LIN {X 0,Y 496.772,Z 250.855,A -85,B 0,C 180,E1 18209.944,E2 18209.944} C_VEL
LIN {X 0,Y 496.758,Z 250.853,A -85,B 0,C 180,E1 18206.403,E2 18206.403} C_VEL
LIN {X 0,Y 496.769,Z 250.851,A -85,B 0,C 180,E1 18202.804,E2 18202.804} C_VEL
LIN {X 0,Y 496.753,Z 250.856,A -85,B 0,C 180,E1 18199.264,E2 18199.264} C_VEL
LIN {X 0,Y 496.754,Z 250.857,A -85,B 0,C 180,E1 18195.648,E2 18195.648} C_VEL
LIN {X 0,Y 496.767,Z 250.857,A -85,B 0,C 180,E1 18192.084,E2 18192.084} C_VEL
LIN {X 0,Y 496.769,Z 250.855,A -85,B 0,C 180,E1 18188.45,E2 18188.45} C_VEL
LIN {X 0,Y 496.745,Z 250.851,A -85,B 0,C 180,E1 18184.966,E2 18184.966} C_VEL
LIN {X 0,Y 496.736,Z 250.854,A -85,B 0,C 180,E1 18181.385,E2 18181.385} C_VEL
LIN {X 0,Y 496.764,Z 250.853,A -85,B 0,C 180,E1 18177.925,E2 18177.925} C_VEL
LIN {X 0,Y 496.768,Z 250.855,A -85,B 0,C 180,E1 18174.341,E2 18174.341} C_VEL
LIN {X 0,Y 496.725,Z 250.858,A -85,B 0,C 180,E1 18170.968,E2 18170.968} C_VEL
LIN {X 0,Y 496.723,Z 250.861,A -85,B 0,C 180,E1 18167.327,E2 18167.327} C_VEL
LIN {X 0,Y 496.769,Z 250.856,A -85,B 0,C 180,E1 18163.995,E2 18163.995} C_VEL
LIN {X 0,Y 496.736,Z 250.862,A -85,B 0,C 180,E1 18160.481,E2 18160.481} C_VEL
LIN {X 0,Y 496.706,Z 250.846,A -85,B 0,C 180,E1 18157.015,E2 18157.015} C_VEL
LIN {X 0,Y 496.788,Z 251.097,A -85,B 0,C 180,E1 18155.823,E2 18155.823} C_VEL
LIN {X 0,Y 498.222,Z 254.643,A -85,B 0,C 180,E1 18155.266,E2 18155.266} C_VEL
LIN {X 0,Y 505.949,Z 273.047,A -85,B 0,C 180,E1 18152.712,E2 18152.712} C_VEL
LIN {X 0,Y 509.561,Z 282.883,A -85,B 0,C 180,E1 18151.46,E2 18151.46} C_VEL
LIN {X 0,Y 508.599,Z 300.101,A -85,B 0,C 180,E1 18150.013,E2 18150.013} C_VEL
LIN {X 0,Y 512.119,Z 319.644,A -85,B 0,C 180,E1 18149.37,E2 18149.37} C_VEL
LIN {X 0,Y 509.717,Z 467.45,A -85,B 0,C 180,E1 18147.041,E2 18147.041} C_VEL
LIN {X 0,Y 508.732,Z 475.141,A -85,B 0,C 180,E1 18146.984,E2 18146.984} C_VEL
LIN {X 0,Y 503.194,Z 495.645,A -85,B 0,C 180,E1 18147.05,E2 18147.05} C_VEL
LIN {X 0,Y 502.468,Z 502.242,A -85,B 0,C 180,E1 18146.991,E2 18146.991} C_VEL
LIN {X 0,Y 501.359,Z 564.042,A -85,B 0,C 180,E1 18145.978,E2 18145.978} C_VEL
LIN {X 0,Y 500.552,Z 584.976,A -85,B 0,C 180,E1 18145.421,E2 18145.421} C_VEL
LIN {X 0,Y 499.562,Z 604.152,A -85,B 0,C 180,E1 18144.698,E2 18144.698} C_VEL
LIN {X 0,Y 498.327,Z 623.36,A -85,B 0,C 180,E1 18143.765,E2 18143.765} C_VEL
LIN {X 0,Y 496.896,Z 642.75,A -85,B 0,C 180,E1 18142.579,E2 18142.579} C_VEL
LIN {X 0,Y 495.485,Z 660.162,A -85,B 0,C 180,E1 18141.279,E2 18141.279} C_VEL
LIN {X 0,Y 494.046,Z 676.802,A -85,B 0,C 180,E1 18139.792,E2 18139.792} C_VEL
LIN {X 0,Y 492.609,Z 692.858,A -85,B 0,C 180,E1 18138.074,E2 18138.074} C_VEL
LIN {X 0,Y 491.318,Z 707.439,A -85,B 0,C 180,E1 18136.22,E2 18136.22} C_VEL
LIN {X 0,Y 490.214,Z 720.639,A -85,B 0,C 180,E1 18134.232,E2 18134.232} C_VEL
LIN {X 0,Y 489.314,Z 733.716,A -85,B 0,C 180,E1 18131.928,E2 18131.928} C_VEL
LIN {X 0,Y 488.706,Z 744.41,A -85,B 0,C 180,E1 18129.668,E2 18129.668} C_VEL
LIN {X 0,Y 488.303,Z 753.506,A -85,B 0,C 180,E1 18127.309,E2 18127.309} C_VEL
LIN {X 0,Y 488.069,Z 760.637,A -85,B 0,C 180,E1 18124.974,E2 18124.974} C_VEL
LIN {X 0,Y 487.961,Z 766.109,A -85,B 0,C 180,E1 18122.61,E2 18122.61} C_VEL
LIN {X 0,Y 487.919,Z 769.788,A -85,B 0,C 180,E1 18120.273,E2 18120.273} C_VEL
LIN {X 0,Y 487.914,Z 771.861,A -85,B 0,C 180,E1 18117.97,E2 18117.97} C_VEL
LIN {X 0,Y 487.908,Z 772.443,A -85,B 0,C 180,E1 18115.621,E2 18115.621} C_VEL
LIN {X 0,Y 487.916,Z 771.488,A -85,B 0,C 180,E1 18113.298,E2 18113.298} C_VEL
LIN {X 0,Y 487.926,Z 768.745,A -85,B 0,C 180,E1 18110.868,E2 18110.868} C_VEL
LIN {X 0,Y 487.978,Z 764.447,A -85,B 0,C 180,E1 18108.518,E2 18108.518} C_VEL
LIN {X 0,Y 488.144,Z 758.138,A -85,B 0,C 180,E1 18106.054,E2 18106.054} C_VEL
LIN {X 0,Y 488.428,Z 750.424,A -85,B 0,C 180,E1 18103.738,E2 18103.738} C_VEL
LIN {X 0,Y 488.861,Z 741.482,A -85,B 0,C 180,E1 18101.564,E2 18101.564} C_VEL
LIN {X 0,Y 489.546,Z 730.05,A -85,B 0,C 180,E1 18099.286,E2 18099.286} C_VEL
LIN {X 0,Y 490.601,Z 715.79,A -85,B 0,C 180,E1 18096.907,E2 18096.907} C_VEL
LIN {X 0,Y 491.817,Z 701.453,A -85,B 0,C 180,E1 18094.899,E2 18094.899} C_VEL
LIN {X 0,Y 493.162,Z 685.95,A -85,B 0,C 180,E1 18093.081,E2 18093.081} C_VEL
LIN {X 0,Y 494.552,Z 669.994,A -85,B 0,C 180,E1 18091.507,E2 18091.507} C_VEL
LIN {X 0,Y 495.957,Z 653.26,A -85,B 0,C 180,E1 18090.117,E2 18090.117} C_VEL
LIN {X 0,Y 497.377,Z 634.922,A -85,B 0,C 180,E1 18088.849,E2 18088.849} C_VEL
LIN {X 0,Y 498.675,Z 616.606,A -85,B 0,C 180,E1 18087.818,E2 18087.818} C_VEL
LIN {X 0,Y 499.814,Z 596.729,A -85,B 0,C 180,E1 18086.934,E2 18086.934} C_VEL
LIN {X 0,Y 500.752,Z 576.616,A -85,B 0,C 180,E1 18086.273,E2 18086.273} C_VEL
LIN {X 0,Y 501.378,Z 555.957,A -85,B 0,C 180,E1 18085.807,E2 18085.807} C_VEL
LIN {X 0,Y 505.231,Z 320.117,A -85,B 0,C 180,E1 18082.071,E2 18082.071} C_VEL
LIN {X 0,Y 501.409,Z 299.001,A -85,B 0,C 180,E1 18081.342,E2 18081.342} C_VEL
LIN {X 0,Y 502.22,Z 285.202,A -85,B 0,C 180,E1 18080.143,E2 18080.143} C_VEL
LIN {X 0,Y 494.741,Z 266.119,A -85,B 0,C 180,E1 18077.631,E2 18077.631} C_VEL
LIN {X 0,Y 488.853,Z 252.1,A -85,B 0,C 180,E1 18075.612,E2 18075.612} C_VEL
LIN {X 0,Y 488.818,Z 251.843,A -85,B 0,C 180,E1 18073.595,E2 18073.595} C_VEL
LIN {X 0,Y 488.826,Z 251.834,A -85,B 0,C 180,E1 18070.028,E2 18070.028} C_VEL
LIN {X 0,Y 488.824,Z 251.807,A -85,B 0,C 180,E1 18066.367,E2 18066.367} C_VEL
LIN {X 0,Y 488.822,Z 251.844,A -85,B 0,C 180,E1 18062.732,E2 18062.732} C_VEL
LIN {X 0,Y 488.81,Z 251.842,A -85,B 0,C 180,E1 18059.11,E2 18059.11} C_VEL
LIN {X 0,Y 488.822,Z 251.842,A -85,B 0,C 180,E1 18055.489,E2 18055.489} C_VEL
LIN {X 0,Y 488.827,Z 251.847,A -85,B 0,C 180,E1 18051.852,E2 18051.852} C_VEL
LIN {X 0,Y 488.831,Z 251.841,A -85,B 0,C 180,E1 18048.292,E2 18048.292} C_VEL
LIN {X 0,Y 488.81,Z 251.841,A -85,B 0,C 180,E1 18044.718,E2 18044.718} C_VEL
LIN {X 0,Y 488.819,Z 251.833,A -85,B 0,C 180,E1 18041.175,E2 18041.175} C_VEL
LIN {X 0,Y 488.828,Z 251.845,A -85,B 0,C 180,E1 18037.67,E2 18037.67} C_VEL
LIN {X 0,Y 488.825,Z 251.839,A -85,B 0,C 180,E1 18034.069,E2 18034.069} C_VEL
LIN {X 0,Y 488.808,Z 251.833,A -85,B 0,C 180,E1 18030.481,E2 18030.481} C_VEL
LIN {X 0,Y 488.813,Z 251.841,A -85,B 0,C 180,E1 18026.874,E2 18026.874} C_VEL
LIN {X 0,Y 488.832,Z 251.841,A -85,B 0,C 180,E1 18023.25,E2 18023.25} C_VEL
LIN {X 0,Y 488.828,Z 251.829,A -85,B 0,C 180,E1 18019.598,E2 18019.598} C_VEL
LIN {X 0,Y 488.812,Z 251.841,A -85,B 0,C 180,E1 18016.029,E2 18016.029} C_VEL
LIN {X 0,Y 488.804,Z 251.844,A -85,B 0,C 180,E1 18012.401,E2 18012.401} C_VEL
LIN {X 0,Y 488.821,Z 251.832,A -85,B 0,C 180,E1 18008.823,E2 18008.823} C_VEL
LIN {X 0,Y 488.829,Z 251.844,A -85,B 0,C 180,E1 18005.28,E2 18005.28} C_VEL
LIN {X 0,Y 488.822,Z 251.835,A -85,B 0,C 180,E1 18001.64,E2 18001.64} C_VEL
LIN {X 0,Y 488.802,Z 251.832,A -85,B 0,C 180,E1 17998.124,E2 17998.124} C_VEL
LIN {X 0,Y 488.82,Z 251.845,A -85,B 0,C 180,E1 17994.6,E2 17994.6} C_VEL
LIN {X 0,Y 488.83,Z 251.837,A -85,B 0,C 180,E1 17991.056,E2 17991.056} C_VEL
LIN {X 0,Y 488.814,Z 251.829,A -85,B 0,C 180,E1 17987.477,E2 17987.477} C_VEL
LIN {X 0,Y 488.8,Z 251.839,A -85,B 0,C 180,E1 17983.969,E2 17983.969} C_VEL
LIN {X 0,Y 488.82,Z 251.845,A -85,B 0,C 180,E1 17980.399,E2 17980.399} C_VEL
LIN {X 0,Y 488.832,Z 251.844,A -85,B 0,C 180,E1 17976.876,E2 17976.876} C_VEL
LIN {X 0,Y 488.815,Z 251.844,A -85,B 0,C 180,E1 17973.255,E2 17973.255} C_VEL
LIN {X 0,Y 488.799,Z 251.848,A -85,B 0,C 180,E1 17969.676,E2 17969.676} C_VEL
LIN {X 0,Y 488.817,Z 251.847,A -85,B 0,C 180,E1 17966.143,E2 17966.143} C_VEL
LIN {X 0,Y 488.833,Z 251.84,A -85,B 0,C 180,E1 17962.522,E2 17962.522} C_VEL
LIN {X 0,Y 488.819,Z 251.84,A -85,B 0,C 180,E1 17958.959,E2 17958.959} C_VEL
LIN {X 0,Y 488.808,Z 251.913,A -85,B 0,C 180,E1 17955.549,E2 17955.549} C_VEL
LIN {X 0,Y 489.229,Z 253.594,A -85,B 0,C 180,E1 17955.245,E2 17955.245} C_VEL
LIN {X 0,Y 492.865,Z 260.965,A -85,B 0,C 180,E1 17954.253,E2 17954.253} C_VEL
LIN {X 0,Y 501.354,Z 279.391,A -85,B 0,C 180,E1 17951.937,E2 17951.937} C_VEL
LIN {X 0,Y 506.352,Z 291.141,A -85,B 0,C 180,E1 17950.588,E2 17950.588} C_VEL
LIN {X 0,Y 505.835,Z 302.61,A -85,B 0,C 180,E1 17949.815,E2 17949.815} C_VEL
LIN {X 0,Y 509.159,Z 324.69,A -85,B 0,C 180,E1 17949.147,E2 17949.147} C_VEL
LIN {X 0,Y 505.913,Z 541.603,A -85,B 0,C 180,E1 17945.733,E2 17945.733} C_VEL
LIN {X 0,Y 504.85,Z 609.184,A -85,B 0,C 180,E1 17944.654,E2 17944.654} C_VEL
LIN {X 0,Y 503.96,Z 630.518,A -85,B 0,C 180,E1 17944.117,E2 17944.117} C_VEL
LIN {X 0,Y 502.77,Z 653.144,A -85,B 0,C 180,E1 17943.329,E2 17943.329} C_VEL
LIN {X 0,Y 501.528,Z 673.269,A -85,B 0,C 180,E1 17942.429,E2 17942.429} C_VEL
LIN {X 0,Y 500.051,Z 692.001,A -85,B 0,C 180,E1 17941.373,E2 17941.373} C_VEL
LIN {X 0,Y 498.309,Z 712.512,A -85,B 0,C 180,E1 17939.973,E2 17939.973} C_VEL
LIN {X 0,Y 496.643,Z 730.768,A -85,B 0,C 180,E1 17938.497,E2 17938.497} C_VEL
LIN {X 0,Y 494.933,Z 748.878,A -85,B 0,C 180,E1 17936.757,E2 17936.757} C_VEL
LIN {X 0,Y 493.327,Z 765.681,A -85,B 0,C 180,E1 17934.868,E2 17934.868} C_VEL
LIN {X 0,Y 491.919,Z 781.186,A -85,B 0,C 180,E1 17932.842,E2 17932.842} C_VEL
LIN {X 0,Y 490.705,Z 795.639,A -85,B 0,C 180,E1 17930.639,E2 17930.639} C_VEL
LIN {X 0,Y 489.724,Z 808.46,A -85,B 0,C 180,E1 17928.324,E2 17928.324} C_VEL
LIN {X 0,Y 488.981,Z 819.817,A -85,B 0,C 180,E1 17925.901,E2 17925.901} C_VEL
LIN {X 0,Y 488.485,Z 829.264,A -85,B 0,C 180,E1 17923.492,E2 17923.492} C_VEL
LIN {X 0,Y 488.176,Z 836.886,A -85,B 0,C 180,E1 17921.099,E2 17921.099} C_VEL
LIN {X 0,Y 488.003,Z 843.148,A -85,B 0,C 180,E1 17918.601,E2 17918.601} C_VEL
LIN {X 0,Y 487.936,Z 847.824,A -85,B 0,C 180,E1 17916.116,E2 17916.116} C_VEL
LIN {X 0,Y 487.907,Z 850.804,A -85,B 0,C 180,E1 17913.625,E2 17913.625} C_VEL
LIN {X 0,Y 487.911,Z 852.305,A -85,B 0,C 180,E1 17911.056,E2 17911.056} C_VEL
LIN {X 0,Y 487.906,Z 852.258,A -85,B 0,C 180,E1 17908.707,E2 17908.707} C_VEL
LIN {X 0,Y 487.908,Z 850.67,A -85,B 0,C 180,E1 17906.239,E2 17906.239} C_VEL
LIN {X 0,Y 487.938,Z 847.63,A -85,B 0,C 180,E1 17903.764,E2 17903.764} C_VEL
LIN {X 0,Y 488.004,Z 843.142,A -85,B 0,C 180,E1 17901.397,E2 17901.397} C_VEL
LIN {X 0,Y 488.184,Z 836.668,A -85,B 0,C 180,E1 17898.828,E2 17898.828} C_VEL
LIN {X 0,Y 488.509,Z 828.845,A -85,B 0,C 180,E1 17896.385,E2 17896.385} C_VEL
LIN {X 0,Y 489.028,Z 819.123,A -85,B 0,C 180,E1 17893.936,E2 17893.936} C_VEL
LIN {X 0,Y 489.771,Z 807.812,A -85,B 0,C 180,E1 17891.552,E2 17891.552} C_VEL
LIN {X 0,Y 490.706,Z 795.623,A -85,B 0,C 180,E1 17889.358,E2 17889.358} C_VEL
LIN {X 0,Y 491.921,Z 781.168,A -85,B 0,C 180,E1 17887.155,E2 17887.155} C_VEL
LIN {X 0,Y 493.328,Z 765.66,A -85,B 0,C 180,E1 17885.129,E2 17885.129} C_VEL
LIN {X 0,Y 494.949,Z 748.687,A -85,B 0,C 180,E1 17883.224,E2 17883.224} C_VEL
LIN {X 0,Y 496.646,Z 730.741,A -85,B 0,C 180,E1 17881.501,E2 17881.501} C_VEL
LIN {X 0,Y 498.312,Z 712.484,A -85,B 0,C 180,E1 17880.024,E2 17880.024} C_VEL
LIN {X 0,Y 500.053,Z 691.996,A -85,B 0,C 180,E1 17878.626,E2 17878.626} C_VEL
LIN {X 0,Y 501.531,Z 673.215,A -85,B 0,C 180,E1 17877.568,E2 17877.568} C_VEL
LIN {X 0,Y 502.804,Z 652.224,A -85,B 0,C 180,E1 17876.637,E2 17876.637} C_VEL
LIN {X 0,Y 503.967,Z 629.777,A -85,B 0,C 180,E1 17875.868,E2 17875.868} C_VEL
LIN {X 0,Y 504.829,Z 608.318,A -85,B 0,C 180,E1 17875.337,E2 17875.337} C_VEL
LIN {X 0,Y 506.756,Z 476.023,A -85,B 0,C 180,E1 17873.262,E2 17873.262} C_VEL
LIN {X 0,Y 508.836,Z 322.634,A -85,B 0,C 180,E1 17870.839,E2 17870.839} C_VEL
LIN {X 0,Y 505.54,Z 301.596,A -85,B 0,C 180,E1 17870.184,E2 17870.184} C_VEL
LIN {X 0,Y 505.959,Z 290.005,A -85,B 0,C 180,E1 17869.363,E2 17869.363} C_VEL
LIN {X 0,Y 495.083,Z 265.808,A -85,B 0,C 180,E1 17866.472,E2 17866.472} C_VEL
LIN {X 0,Y 490.052,Z 255.211,A -85,B 0,C 180,E1 17865.072,E2 17865.072} C_VEL
LIN {X 0,Y 488.846,Z 252.112,A -85,B 0,C 180,E1 17864.619,E2 17864.619} C_VEL
LIN {X 0,Y 488.829,Z 251.842,A -85,B 0,C 180,E1 17861.508,E2 17861.508} C_VEL
LIN {X 0,Y 488.83,Z 251.844,A -85,B 0,C 180,E1 17857.852,E2 17857.852} C_VEL
LIN {X 0,Y 488.82,Z 251.844,A -85,B 0,C 180,E1 17854.229,E2 17854.229} C_VEL
LIN {X 0,Y 488.818,Z 251.844,A -85,B 0,C 180,E1 17850.619,E2 17850.619} C_VEL
LIN {X 0,Y 488.829,Z 251.841,A -85,B 0,C 180,E1 17847.007,E2 17847.007} C_VEL
LIN {X 0,Y 488.816,Z 251.841,A -85,B 0,C 180,E1 17843.38,E2 17843.38} C_VEL
LIN {X 0,Y 488.823,Z 251.844,A -85,B 0,C 180,E1 17839.795,E2 17839.795} C_VEL
LIN {X 0,Y 488.828,Z 251.844,A -85,B 0,C 180,E1 17836.152,E2 17836.152} C_VEL
LIN {X 0,Y 488.83,Z 251.844,A -85,B 0,C 180,E1 17832.523,E2 17832.523} C_VEL
LIN {X 0,Y 488.815,Z 251.843,A -85,B 0,C 180,E1 17828.895,E2 17828.895} C_VEL
LIN {X 0,Y 488.801,Z 251.843,A -85,B 0,C 180,E1 17825.4,E2 17825.4} C_VEL
LIN {X 0,Y 488.823,Z 251.841,A -85,B 0,C 180,E1 17821.876,E2 17821.876} C_VEL
LIN {X 0,Y 488.831,Z 251.839,A -85,B 0,C 180,E1 17818.36,E2 17818.36} C_VEL
LIN {X 0,Y 488.797,Z 251.845,A -85,B 0,C 180,E1 17814.837,E2 17814.837} C_VEL
LIN {X 0,Y 488.787,Z 251.849,A -85,B 0,C 180,E1 17811.295,E2 17811.295} C_VEL
LIN {X 0,Y 488.818,Z 251.843,A -85,B 0,C 180,E1 17807.839,E2 17807.839} C_VEL
LIN {X 0,Y 488.818,Z 251.848,A -85,B 0,C 180,E1 17804.337,E2 17804.337} C_VEL
LIN {X 0,Y 488.776,Z 251.852,A -85,B 0,C 180,E1 17800.896,E2 17800.896} C_VEL
LIN {X 0,Y 488.771,Z 251.834,A -85,B 0,C 180,E1 17797.256,E2 17797.256} C_VEL
LIN {X 0,Y 488.823,Z 252.135,A -85,B 0,C 180,E1 17796.59,E2 17796.59} C_VEL
LIN {X 0,Y 495.725,Z 268.342,A -85,B 0,C 180,E1 17794.174,E2 17794.174} C_VEL
LIN {X 0,Y 502.718,Z 285.823,A -85,B 0,C 180,E1 17791.814,E2 17791.814} C_VEL
LIN {X 0,Y 501.902,Z 300.091,A -85,B 0,C 180,E1 17790.599,E2 17790.599} C_VEL
LIN {X 0,Y 505.67,Z 321.039,A -85,B 0,C 180,E1 17789.889,E2 17789.889} C_VEL
LIN {X 0,Y 502.468,Z 502.242,A -85,B 0,C 180,E1 17786.991,E2 17786.991} C_VEL
LIN {X 0,Y 501.504,Z 509.932,A -85,B 0,C 180,E1 17786.932,E2 17786.932} C_VEL
LIN {X 0,Y 495.893,Z 530.424,A -85,B 0,C 180,E1 17787.002,E2 17787.002} C_VEL
LIN {X 0,Y 495.165,Z 537.023,A -85,B 0,C 180,E1 17786.942,E2 17786.942} C_VEL
LIN {X 0,Y 494.491,Z 566.986,A -85,B 0,C 180,E1 17786.409,E2 17786.409} C_VEL
LIN {X 0,Y 493.652,Z 587.312,A -85,B 0,C 180,E1 17785.84,E2 17785.84} C_VEL
LIN {X 0,Y 492.563,Z 606.745,A -85,B 0,C 180,E1 17785.082,E2 17785.082} C_VEL
LIN {X 0,Y 491.214,Z 625.979,A -85,B 0,C 180,E1 17784.109,E2 17784.109} C_VEL
LIN {X 0,Y 489.754,Z 644.17,A -85,B 0,C 180,E1 17782.964,E2 17782.964} C_VEL
LIN {X 0,Y 488.174,Z 662.153,A -85,B 0,C 180,E1 17781.585,E2 17781.585} C_VEL
LIN {X 0,Y 486.698,Z 677.989,A -85,B 0,C 180,E1 17780.138,E2 17780.138} C_VEL
LIN {X 0,Y 485.179,Z 693.746,A -85,B 0,C 180,E1 17778.425,E2 17778.425} C_VEL
LIN {X 0,Y 483.783,Z 708.188,A -85,B 0,C 180,E1 17776.559,E2 17776.559} C_VEL
LIN {X 0,Y 482.576,Z 721.36,A -85,B 0,C 180,E1 17774.544,E2 17774.544} C_VEL
LIN {X 0,Y 481.576,Z 733.418,A -85,B 0,C 180,E1 17772.345,E2 17772.345} C_VEL
LIN {X 0,Y 480.795,Z 744.555,A -85,B 0,C 180,E1 17769.884,E2 17769.884} C_VEL
LIN {X 0,Y 480.337,Z 753.727,A -85,B 0,C 180,E1 17767.433,E2 17767.433} C_VEL
LIN {X 0,Y 480.083,Z 760.779,A -85,B 0,C 180,E1 17765.069,E2 17765.069} C_VEL
LIN {X 0,Y 479.968,Z 766.157,A -85,B 0,C 180,E1 17762.693,E2 17762.693} C_VEL
LIN {X 0,Y 479.921,Z 769.878,A -85,B 0,C 180,E1 17760.278,E2 17760.278} C_VEL
LIN {X 0,Y 479.914,Z 771.889,A -85,B 0,C 180,E1 17757.953,E2 17757.953} C_VEL
LIN {X 0,Y 479.908,Z 772.43,A -85,B 0,C 180,E1 17755.549,E2 17755.549} C_VEL
LIN {X 0,Y 479.918,Z 771.439,A -85,B 0,C 180,E1 17753.19,E2 17753.19} C_VEL
LIN {X 0,Y 479.927,Z 768.645,A -85,B 0,C 180,E1 17750.708,E2 17750.708} C_VEL
LIN {X 0,Y 479.992,Z 764.32,A -85,B 0,C 180,E1 17748.334,E2 17748.334} C_VEL
LIN {X 0,Y 480.173,Z 758.026,A -85,B 0,C 180,E1 17745.849,E2 17745.849} C_VEL
LIN {X 0,Y 480.497,Z 750.218,A -85,B 0,C 180,E1 17743.478,E2 17743.478} C_VEL
LIN {X 0,Y 481.102,Z 739.711,A -85,B 0,C 180,E1 17740.903,E2 17740.903} C_VEL
LIN {X 0,Y 481.916,Z 728.949,A -85,B 0,C 180,E1 17738.713,E2 17738.713} C_VEL
LIN {X 0,Y 482.944,Z 716.915,A -85,B 0,C 180,E1 17736.659,E2 17736.659} C_VEL
LIN {X 0,Y 484.254,Z 702.628,A -85,B 0,C 180,E1 17734.62,E2 17734.62} C_VEL
LIN {X 0,Y 485.647,Z 687.74,A -85,B 0,C 180,E1 17732.833,E2 17732.833} C_VEL
LIN {X 0,Y 487.138,Z 672.001,A -85,B 0,C 180,E1 17731.236,E2 17731.236} C_VEL
LIN {X 0,Y 488.768,Z 654.028,A -85,B 0,C 180,E1 17729.708,E2 17729.708} C_VEL
LIN {X 0,Y 490.291,Z 635.723,A -85,B 0,C 180,E1 17728.424,E2 17728.424} C_VEL
LIN {X 0,Y 491.68,Z 617.468,A -85,B 0,C 180,E1 17727.379,E2 17727.379} C_VEL
LIN {X 0,Y 492.891,Z 597.642,A -85,B 0,C 180,E1 17726.483,E2 17726.483} C_VEL
LIN {X 0,Y 493.89,Z 577.709,A -85,B 0,C 180,E1 17725.815,E2 17725.815} C_VEL
LIN {X 0,Y 494.571,Z 556.973,A -85,B 0,C 180,E1 17725.334,E2 17725.334} C_VEL
LIN {X 0,Y 498.755,Z 321.538,A -85,B 0,C 180,E1 17721.55,E2 17721.55} C_VEL
LIN {X 0,Y 494.681,Z 298.995,A -85,B 0,C 180,E1 17720.755,E2 17720.755} C_VEL
LIN {X 0,Y 495.303,Z 288.494,A -85,B 0,C 180,E1 17719.828,E2 17719.828} C_VEL
LIN {X 0,Y 488.224,Z 270.414,A -85,B 0,C 180,E1 17717.404,E2 17717.404} C_VEL
LIN {X 0,Y 482.117,Z 256.202,A -85,B 0,C 180,E1 17715.345,E2 17715.345} C_VEL
LIN {X 0,Y 480.906,Z 252.954,A -85,B 0,C 180,E1 17714.815,E2 17714.815} C_VEL
LIN {X 0,Y 480.871,Z 252.801,A -85,B 0,C 180,E1 17711.2,E2 17711.2} C_VEL
LIN {X 0,Y 480.884,Z 252.808,A -85,B 0,C 180,E1 17707.637,E2 17707.637} C_VEL
LIN {X 0,Y 480.888,Z 252.828,A -85,B 0,C 180,E1 17703.98,E2 17703.98} C_VEL
LIN {X 0,Y 480.892,Z 252.831,A -85,B 0,C 180,E1 17700.342,E2 17700.342} C_VEL
LIN {X 0,Y 480.88,Z 252.833,A -85,B 0,C 180,E1 17696.701,E2 17696.701} C_VEL
LIN {X 0,Y 480.873,Z 252.835,A -85,B 0,C 180,E1 17693.067,E2 17693.067} C_VEL
LIN {X 0,Y 480.892,Z 252.824,A -85,B 0,C 180,E1 17689.548,E2 17689.548} C_VEL
LIN {X 0,Y 480.887,Z 252.822,A -85,B 0,C 180,E1 17685.853,E2 17685.853} C_VEL
LIN {X 0,Y 480.89,Z 252.828,A -85,B 0,C 180,E1 17682.187,E2 17682.187} C_VEL
LIN {X 0,Y 480.87,Z 252.832,A -85,B 0,C 180,E1 17678.577,E2 17678.577} C_VEL
LIN {X 0,Y 480.871,Z 252.83,A -85,B 0,C 180,E1 17674.874,E2 17674.874} C_VEL
LIN {X 0,Y 480.892,Z 252.821,A -85,B 0,C 180,E1 17671.294,E2 17671.294} C_VEL
LIN {X 0,Y 480.891,Z 252.833,A -85,B 0,C 180,E1 17667.622,E2 17667.622} C_VEL
LIN {X 0,Y 480.882,Z 252.824,A -85,B 0,C 180,E1 17664.048,E2 17664.048} C_VEL
LIN {X 0,Y 480.865,Z 252.822,A -85,B 0,C 180,E1 17660.444,E2 17660.444} C_VEL
LIN {X 0,Y 480.877,Z 252.835,A -85,B 0,C 180,E1 17656.798,E2 17656.798} C_VEL
LIN {X 0,Y 480.889,Z 252.817,A -85,B 0,C 180,E1 17653.22,E2 17653.22} C_VEL
LIN {X 0,Y 480.89,Z 252.827,A -85,B 0,C 180,E1 17649.574,E2 17649.574} C_VEL
LIN {X 0,Y 480.87,Z 252.832,A -85,B 0,C 180,E1 17645.966,E2 17645.966} C_VEL
LIN {X 0,Y 480.865,Z 252.825,A -85,B 0,C 180,E1 17642.382,E2 17642.382} C_VEL
LIN {X 0,Y 480.887,Z 252.826,A -85,B 0,C 180,E1 17638.808,E2 17638.808} C_VEL
LIN {X 0,Y 480.891,Z 252.83,A -85,B 0,C 180,E1 17635.228,E2 17635.228} C_VEL
LIN {X 0,Y 480.873,Z 252.824,A -85,B 0,C 180,E1 17631.63,E2 17631.63} C_VEL
LIN {X 0,Y 480.862,Z 252.82,A -85,B 0,C 180,E1 17627.998,E2 17627.998} C_VEL
LIN {X 0,Y 480.882,Z 252.83,A -85,B 0,C 180,E1 17624.441,E2 17624.441} C_VEL
LIN {X 0,Y 480.892,Z 252.834,A -85,B 0,C 180,E1 17620.821,E2 17620.821} C_VEL
LIN {X 0,Y 480.883,Z 252.831,A -85,B 0,C 180,E1 17617.248,E2 17617.248} C_VEL
LIN {X 0,Y 480.863,Z 252.835,A -85,B 0,C 180,E1 17613.656,E2 17613.656} C_VEL
LIN {X 0,Y 480.871,Z 252.837,A -85,B 0,C 180,E1 17610.064,E2 17610.064} C_VEL
LIN {X 0,Y 480.893,Z 252.835,A -85,B 0,C 180,E1 17606.482,E2 17606.482} C_VEL
LIN {X 0,Y 480.888,Z 252.834,A -85,B 0,C 180,E1 17602.917,E2 17602.917} C_VEL
LIN {X 0,Y 480.86,Z 252.829,A -85,B 0,C 180,E1 17599.369,E2 17599.369} C_VEL
LIN {X 0,Y 480.907,Z 252.932,A -85,B 0,C 180,E1 17596.344,E2 17596.344} C_VEL
LIN {X 0,Y 481.44,Z 254.914,A -85,B 0,C 180,E1 17595.997,E2 17595.997} C_VEL
LIN {X 0,Y 486.703,Z 265.481,A -85,B 0,C 180,E1 17594.532,E2 17594.532} C_VEL
LIN {X 0,Y 495.574,Z 285.003,A -85,B 0,C 180,E1 17592.052,E2 17592.052} C_VEL
LIN {X 0,Y 499.604,Z 294.361,A -85,B 0,C 180,E1 17590.95,E2 17590.95} C_VEL
LIN {X 0,Y 499.25,Z 302.656,A -85,B 0,C 180,E1 17590.394,E2 17590.394} C_VEL
LIN {X 0,Y 502.723,Z 326.091,A -85,B 0,C 180,E1 17589.671,E2 17589.671} C_VEL
LIN {X 0,Y 499.208,Z 542.708,A -85,B 0,C 180,E1 17586.22,E2 17586.22} C_VEL
LIN {X 0,Y 498.08,Z 608.856,A -85,B 0,C 180,E1 17585.151,E2 17585.151} C_VEL
LIN {X 0,Y 497.137,Z 630.034,A -85,B 0,C 180,E1 17584.612,E2 17584.612} C_VEL
LIN {X 0,Y 495.846,Z 652.722,A -85,B 0,C 180,E1 17583.815,E2 17583.815} C_VEL
LIN {X 0,Y 494.473,Z 673.295,A -85,B 0,C 180,E1 17582.881,E2 17582.881} C_VEL
LIN {X 0,Y 492.888,Z 692.996,A -85,B 0,C 180,E1 17581.768,E2 17581.768} C_VEL
LIN {X 0,Y 491.157,Z 713.181,A -85,B 0,C 180,E1 17580.394,E2 17580.394} C_VEL
LIN {X 0,Y 489.453,Z 730.766,A -85,B 0,C 180,E1 17578.955,E2 17578.955} C_VEL
LIN {X 0,Y 487.609,Z 748.711,A -85,B 0,C 180,E1 17577.209,E2 17577.209} C_VEL
LIN {X 0,Y 485.852,Z 765.68,A -85,B 0,C 180,E1 17575.277,E2 17575.277} C_VEL
LIN {X 0,Y 484.325,Z 781.185,A -85,B 0,C 180,E1 17573.221,E2 17573.221} C_VEL
LIN {X 0,Y 482.995,Z 795.639,A -85,B 0,C 180,E1 17570.984,E2 17570.984} C_VEL
LIN {X 0,Y 481.92,Z 808.458,A -85,B 0,C 180,E1 17568.632,E2 17568.632} C_VEL
LIN {X 0,Y 481.103,Z 819.816,A -85,B 0,C 180,E1 17566.168,E2 17566.168} C_VEL
LIN {X 0,Y 480.544,Z 829.434,A -85,B 0,C 180,E1 17563.669,E2 17563.669} C_VEL
LIN {X 0,Y 480.21,Z 836.901,A -85,B 0,C 180,E1 17561.28,E2 17561.28} C_VEL
LIN {X 0,Y 480.013,Z 843.148,A -85,B 0,C 180,E1 17558.745,E2 17558.745} C_VEL
LIN {X 0,Y 479.939,Z 847.824,A -85,B 0,C 180,E1 17556.218,E2 17556.218} C_VEL
LIN {X 0,Y 479.907,Z 850.788,A -85,B 0,C 180,E1 17553.702,E2 17553.702} C_VEL
LIN {X 0,Y 479.911,Z 852.304,A -85,B 0,C 180,E1 17551.073,E2 17551.073} C_VEL
LIN {X 0,Y 479.906,Z 852.258,A -85,B 0,C 180,E1 17548.686,E2 17548.686} C_VEL
LIN {X 0,Y 479.908,Z 850.67,A -85,B 0,C 180,E1 17546.176,E2 17546.176} C_VEL
LIN {X 0,Y 479.938,Z 847.63,A -85,B 0,C 180,E1 17543.66,E2 17543.66} C_VEL
LIN {X 0,Y 480.013,Z 843.142,A -85,B 0,C 180,E1 17541.253,E2 17541.253} C_VEL
LIN {X 0,Y 480.211,Z 836.877,A -85,B 0,C 180,E1 17538.712,E2 17538.712} C_VEL
LIN {X 0,Y 480.554,Z 829.253,A -85,B 0,C 180,E1 17536.278,E2 17536.278} C_VEL
LIN {X 0,Y 481.104,Z 819.804,A -85,B 0,C 180,E1 17533.829,E2 17533.829} C_VEL
LIN {X 0,Y 481.921,Z 808.446,A -85,B 0,C 180,E1 17531.366,E2 17531.366} C_VEL
LIN {X 0,Y 482.927,Z 796.343,A -85,B 0,C 180,E1 17529.137,E2 17529.137} C_VEL
LIN {X 0,Y 484.153,Z 782.857,A -85,B 0,C 180,E1 17527.025,E2 17527.025} C_VEL
LIN {X 0,Y 485.754,Z 766.673,A -85,B 0,C 180,E1 17524.845,E2 17524.845} C_VEL
LIN {X 0,Y 487.44,Z 750.508,A -85,B 0,C 180,E1 17522.976,E2 17522.976} C_VEL
LIN {X 0,Y 489.183,Z 733.134,A -85,B 0,C 180,E1 17521.265,E2 17521.265} C_VEL
LIN {X 0,Y 491.006,Z 714.881,A -85,B 0,C 180,E1 17519.734,E2 17519.734} C_VEL
LIN {X 0,Y 492.633,Z 696.067,A -85,B 0,C 180,E1 17518.422,E2 17518.422} C_VEL
LIN {X 0,Y 494.252,Z 675.499,A -85,B 0,C 180,E1 17517.246,E2 17517.246} C_VEL
LIN {X 0,Y 495.723,Z 653.82,A -85,B 0,C 180,E1 17516.242,E2 17516.242} C_VEL
LIN {X 0,Y 496.97,Z 632.161,A -85,B 0,C 180,E1 17515.463,E2 17515.463} C_VEL
LIN {X 0,Y 497.884,Z 611.575,A -85,B 0,C 180,E1 17514.927,E2 17514.927} C_VEL
LIN {X 0,Y 498.558,Z 579.593,A -85,B 0,C 180,E1 17514.377,E2 17514.377} C_VEL
LIN {X 0,Y 501.998,Z 355.182,A -85,B 0,C 180,E1 17510.836,E2 17510.836} C_VEL
LIN {X 0,Y 502.297,Z 323.712,A -85,B 0,C 180,E1 17510.313,E2 17510.313} C_VEL
LIN {X 0,Y 498.898,Z 301.444,A -85,B 0,C 180,E1 17509.603,E2 17509.603} C_VEL
LIN {X 0,Y 499.201,Z 293.581,A -85,B 0,C 180,E1 17509.034,E2 17509.034} C_VEL
LIN {X 0,Y 488.331,Z 269.018,A -85,B 0,C 180,E1 17506.043,E2 17506.043} C_VEL
LIN {X 0,Y 482.275,Z 256.458,A -85,B 0,C 180,E1 17504.321,E2 17504.321} C_VEL
LIN {X 0,Y 480.932,Z 253.116,A -85,B 0,C 180,E1 17503.814,E2 17503.814} C_VEL
LIN {X 0,Y 480.891,Z 252.822,A -85,B 0,C 180,E1 17501.868,E2 17501.868} C_VEL
LIN {X 0,Y 480.877,Z 252.833,A -85,B 0,C 180,E1 17498.288,E2 17498.288} C_VEL
LIN {X 0,Y 480.881,Z 252.835,A -85,B 0,C 180,E1 17494.73,E2 17494.73} C_VEL
LIN {X 0,Y 480.892,Z 252.831,A -85,B 0,C 180,E1 17491.06,E2 17491.06} C_VEL
LIN {X 0,Y 480.881,Z 252.833,A -85,B 0,C 180,E1 17487.397,E2 17487.397} C_VEL
LIN {X 0,Y 480.885,Z 252.829,A -85,B 0,C 180,E1 17483.789,E2 17483.789} C_VEL
LIN {X 0,Y 480.888,Z 252.828,A -85,B 0,C 180,E1 17480.191,E2 17480.191} C_VEL
LIN {X 0,Y 480.889,Z 252.829,A -85,B 0,C 180,E1 17476.551,E2 17476.551} C_VEL
LIN {X 0,Y 480.879,Z 252.833,A -85,B 0,C 180,E1 17472.978,E2 17472.978} C_VEL
LIN {X 0,Y 480.865,Z 252.835,A -85,B 0,C 180,E1 17469.335,E2 17469.335} C_VEL
LIN {X 0,Y 480.877,Z 252.834,A -85,B 0,C 180,E1 17465.729,E2 17465.729} C_VEL
LIN {X 0,Y 480.893,Z 252.831,A -85,B 0,C 180,E1 17462.146,E2 17462.146} C_VEL
LIN {X 0,Y 480.88,Z 252.829,A -85,B 0,C 180,E1 17458.571,E2 17458.571} C_VEL
LIN {X 0,Y 480.854,Z 252.834,A -85,B 0,C 180,E1 17454.991,E2 17454.991} C_VEL
LIN {X 0,Y 480.852,Z 252.838,A -85,B 0,C 180,E1 17451.391,E2 17451.391} C_VEL
LIN {X 0,Y 480.882,Z 252.831,A -85,B 0,C 180,E1 17447.879,E2 17447.879} C_VEL
LIN {X 0,Y 480.884,Z 252.837,A -85,B 0,C 180,E1 17444.299,E2 17444.299} C_VEL
LIN {X 0,Y 480.842,Z 252.841,A -85,B 0,C 180,E1 17440.744,E2 17440.744} C_VEL
LIN {X 0,Y 480.87,Z 253.032,A -85,B 0,C 180,E1 17437.437,E2 17437.437} C_VEL
LIN {X 0,Y 482.012,Z 256.119,A -85,B 0,C 180,E1 17436.919,E2 17436.919} C_VEL
LIN {X 0,Y 487.648,Z 268.595,A -85,B 0,C 180,E1 17434.996,E2 17434.996} C_VEL
LIN {X 0,Y 495.308,Z 287.723,A -85,B 0,C 180,E1 17432.337,E2 17432.337} C_VEL
LIN {X 0,Y 495.915,Z 289.453,A -85,B 0,C 180,E1 17432.113,E2 17432.113} C_VEL
LIN {X 0,Y 495.258,Z 300.123,A -85,B 0,C 180,E1 17431.202,E2 17431.202} C_VEL
LIN {X 0,Y 499.269,Z 322.458,A -85,B 0,C 180,E1 17430.421,E2 17430.421} C_VEL
LIN {X 0,Y 495.165,Z 537.023,A -85,B 0,C 180,E1 17426.942,E2 17426.942} C_VEL
LIN {X 0,Y 494.204,Z 544.712,A -85,B 0,C 180,E1 17426.884,E2 17426.884} C_VEL
LIN {X 0,Y 488.667,Z 564.066,A -85,B 0,C 180,E1 17426.931,E2 17426.931} C_VEL
LIN {X 0,Y 487.582,Z 571.681,A -85,B 0,C 180,E1 17426.809,E2 17426.809} C_VEL
LIN {X 0,Y 486.62,Z 592.182,A -85,B 0,C 180,E1 17426.175,E2 17426.175} C_VEL
LIN {X 0,Y 485.373,Z 611.82,A -85,B 0,C 180,E1 17425.352,E2 17425.352} C_VEL
LIN {X 0,Y 484.011,Z 630.169,A -85,B 0,C 180,E1 17424.372,E2 17424.372} C_VEL
LIN {X 0,Y 482.359,Z 648.671,A -85,B 0,C 180,E1 17423.143,E2 17423.143} C_VEL
LIN {X 0,Y 480.693,Z 666.092,A -85,B 0,C 180,E1 17421.732,E2 17421.732} C_VEL
LIN {X 0,Y 478.969,Z 682.84,A -85,B 0,C 180,E1 17420.11,E2 17420.11} C_VEL
LIN {X 0,Y 477.305,Z 698.731,A -85,B 0,C 180,E1 17418.274,E2 17418.274} C_VEL
LIN {X 0,Y 475.829,Z 713.144,A -85,B 0,C 180,E1 17416.291,E2 17416.291} C_VEL
LIN {X 0,Y 474.598,Z 725.859,A -85,B 0,C 180,E1 17414.215,E2 17414.215} C_VEL
LIN {X 0,Y 473.609,Z 737.207,A -85,B 0,C 180,E1 17412.004,E2 17412.004} C_VEL
LIN {X 0,Y 472.866,Z 747.033,A -85,B 0,C 180,E1 17409.679,E2 17409.679} C_VEL
LIN {X 0,Y 472.384,Z 754.836,A -85,B 0,C 180,E1 17407.408,E2 17407.408} C_VEL
LIN {X 0,Y 472.083,Z 761.725,A -85,B 0,C 180,E1 17404.881,E2 17404.881} C_VEL
LIN {X 0,Y 471.951,Z 767.07,A -85,B 0,C 180,E1 17402.269,E2 17402.269} C_VEL
LIN {X 0,Y 471.921,Z 770.417,A -85,B 0,C 180,E1 17399.862,E2 17399.862} C_VEL
LIN {X 0,Y 471.911,Z 772.211,A -85,B 0,C 180,E1 17397.412,E2 17397.412} C_VEL
LIN {X 0,Y 471.911,Z 772.342,A -85,B 0,C 180,E1 17395.073,E2 17395.073} C_VEL
LIN {X 0,Y 471.916,Z 770.862,A -85,B 0,C 180,E1 17392.523,E2 17392.523} C_VEL
LIN {X 0,Y 471.945,Z 767.802,A -85,B 0,C 180,E1 17390.074,E2 17390.074} C_VEL
LIN {X 0,Y 472.036,Z 763.059,A -85,B 0,C 180,E1 17387.608,E2 17387.608} C_VEL
LIN {X 0,Y 472.29,Z 756.63,A -85,B 0,C 180,E1 17385.095,E2 17385.095} C_VEL
LIN {X 0,Y 472.727,Z 748.734,A -85,B 0,C 180,E1 17382.708,E2 17382.708} C_VEL
LIN {X 0,Y 473.413,Z 739.044,A -85,B 0,C 180,E1 17380.343,E2 17380.343} C_VEL
LIN {X 0,Y 474.344,Z 727.994,A -85,B 0,C 180,E1 17378.12,E2 17378.12} C_VEL
LIN {X 0,Y 475.527,Z 715.437,A -85,B 0,C 180,E1 17376.005,E2 17376.005} C_VEL
LIN {X 0,Y 476.895,Z 701.973,A -85,B 0,C 180,E1 17374.089,E2 17374.089} C_VEL
LIN {X 0,Y 478.504,Z 686.356,A -85,B 0,C 180,E1 17372.217,E2 17372.217} C_VEL
LIN {X 0,Y 480.182,Z 669.597,A -85,B 0,C 180,E1 17370.538,E2 17370.538} C_VEL
LIN {X 0,Y 481.813,Z 652.514,A -85,B 0,C 180,E1 17369.109,E2 17369.109} C_VEL
LIN {X 0,Y 483.392,Z 634.641,A -85,B 0,C 180,E1 17367.868,E2 17367.868} C_VEL
LIN {X 0,Y 484.863,Z 615.953,A -85,B 0,C 180,E1 17366.81,E2 17366.81} C_VEL
LIN {X 0,Y 486.152,Z 596.202,A -85,B 0,C 180,E1 17365.927,E2 17365.927} C_VEL
LIN {X 0,Y 487.204,Z 575.869,A -85,B 0,C 180,E1 17365.256,E2 17365.256} C_VEL
LIN {X 0,Y 487.883,Z 555.143,A -85,B 0,C 180,E1 17364.795,E2 17364.795} C_VEL
LIN {X 0,Y 492.319,Z 323.023,A -85,B 0,C 180,E1 17361.019,E2 17361.019} C_VEL
LIN {X 0,Y 488.001,Z 299.219,A -85,B 0,C 180,E1 17360.167,E2 17360.167} C_VEL
LIN {X 0,Y 488.393,Z 291.803,A -85,B 0,C 180,E1 17359.503,E2 17359.503} C_VEL
LIN {X 0,Y 480.817,Z 272.352,A -85,B 0,C 180,E1 17356.839,E2 17356.839} C_VEL
LIN {X 0,Y 474.08,Z 257.02,A -85,B 0,C 180,E1 17354.537,E2 17354.537} C_VEL
LIN {X 0,Y 472.977,Z 254.016,A -85,B 0,C 180,E1 17354.05,E2 17354.05} C_VEL
LIN {X 0,Y 472.947,Z 253.796,A -85,B 0,C 180,E1 17350.488,E2 17350.488} C_VEL
LIN {X 0,Y 472.937,Z 253.783,A -85,B 0,C 180,E1 17346.871,E2 17346.871} C_VEL
LIN {X 0,Y 472.935,Z 253.826,A -85,B 0,C 180,E1 17343.238,E2 17343.238} C_VEL
LIN {X 0,Y 472.951,Z 253.824,A -85,B 0,C 180,E1 17339.6,E2 17339.6} C_VEL
LIN {X 0,Y 472.95,Z 253.825,A -85,B 0,C 180,E1 17335.93,E2 17335.93} C_VEL
LIN {X 0,Y 472.952,Z 253.821,A -85,B 0,C 180,E1 17332.189,E2 17332.189} C_VEL
LIN {X 0,Y 472.941,Z 253.821,A -85,B 0,C 180,E1 17328.571,E2 17328.571} C_VEL
LIN {X 0,Y 472.931,Z 253.818,A -85,B 0,C 180,E1 17324.91,E2 17324.91} C_VEL
LIN {X 0,Y 472.946,Z 253.809,A -85,B 0,C 180,E1 17321.267,E2 17321.267} C_VEL
LIN {X 0,Y 472.951,Z 253.822,A -85,B 0,C 180,E1 17317.658,E2 17317.658} C_VEL
LIN {X 0,Y 472.952,Z 253.817,A -85,B 0,C 180,E1 17313.924,E2 17313.924} C_VEL
LIN {X 0,Y 472.936,Z 253.808,A -85,B 0,C 180,E1 17310.348,E2 17310.348} C_VEL
LIN {X 0,Y 472.931,Z 253.817,A -85,B 0,C 180,E1 17306.763,E2 17306.763} C_VEL
LIN {X 0,Y 472.953,Z 253.821,A -85,B 0,C 180,E1 17303.134,E2 17303.134} C_VEL
LIN {X 0,Y 472.95,Z 253.805,A -85,B 0,C 180,E1 17299.464,E2 17299.464} C_VEL
LIN {X 0,Y 472.948,Z 253.818,A -85,B 0,C 180,E1 17295.825,E2 17295.825} C_VEL
LIN {X 0,Y 472.928,Z 253.82,A -85,B 0,C 180,E1 17292.204,E2 17292.204} C_VEL
LIN {X 0,Y 472.928,Z 253.808,A -85,B 0,C 180,E1 17288.509,E2 17288.509} C_VEL
LIN {X 0,Y 472.95,Z 253.823,A -85,B 0,C 180,E1 17284.971,E2 17284.971} C_VEL
LIN {X 0,Y 472.951,Z 253.814,A -85,B 0,C 180,E1 17281.332,E2 17281.332} C_VEL
LIN {X 0,Y 472.93,Z 253.807,A -85,B 0,C 180,E1 17277.818,E2 17277.818} C_VEL
LIN {X 0,Y 472.925,Z 253.82,A -85,B 0,C 180,E1 17274.175,E2 17274.175} C_VEL
LIN {X 0,Y 472.947,Z 253.821,A -85,B 0,C 180,E1 17270.631,E2 17270.631} C_VEL
LIN {X 0,Y 472.951,Z 253.806,A -85,B 0,C 180,E1 17267.048,E2 17267.048} C_VEL
LIN {X 0,Y 472.931,Z 253.813,A -85,B 0,C 180,E1 17263.542,E2 17263.542} C_VEL
LIN {X 0,Y 472.924,Z 253.819,A -85,B 0,C 180,E1 17259.97,E2 17259.97} C_VEL
LIN {X 0,Y 472.95,Z 253.823,A -85,B 0,C 180,E1 17256.448,E2 17256.448} C_VEL
LIN {X 0,Y 472.956,Z 253.823,A -85,B 0,C 180,E1 17252.829,E2 17252.829} C_VEL
LIN {X 0,Y 472.936,Z 253.824,A -85,B 0,C 180,E1 17249.227,E2 17249.227} C_VEL
LIN {X 0,Y 472.922,Z 253.821,A -85,B 0,C 180,E1 17245.632,E2 17245.632} C_VEL
LIN {X 0,Y 472.935,Z 253.816,A -85,B 0,C 180,E1 17242.032,E2 17242.032} C_VEL
LIN {X 0,Y 472.955,Z 253.823,A -85,B 0,C 180,E1 17238.408,E2 17238.408} C_VEL
LIN {X 0,Y 472.934,Z 253.888,A -85,B 0,C 180,E1 17237.188,E2 17237.188} C_VEL
LIN {X 0,Y 473.323,Z 255.437,A -85,B 0,C 180,E1 17236.892,E2 17236.892} C_VEL
LIN {X 0,Y 479.291,Z 267.509,A -85,B 0,C 180,E1 17235.161,E2 17235.161} C_VEL
LIN {X 0,Y 487.634,Z 285.693,A -85,B 0,C 180,E1 17232.772,E2 17232.772} C_VEL
LIN {X 0,Y 492.847,Z 298.012,A -85,B 0,C 180,E1 17231.291,E2 17231.291} C_VEL
LIN {X 0,Y 492.73,Z 302.817,A -85,B 0,C 180,E1 17230.986,E2 17230.986} C_VEL
LIN {X 0,Y 496.336,Z 327.486,A -85,B 0,C 180,E1 17230.208,E2 17230.208} C_VEL
LIN {X 0,Y 492.544,Z 543.513,A -85,B 0,C 180,E1 17226.724,E2 17226.724} C_VEL
LIN {X 0,Y 491.347,Z 608.508,A -85,B 0,C 180,E1 17225.66,E2 17225.66} C_VEL
LIN {X 0,Y 490.349,Z 629.623,A -85,B 0,C 180,E1 17225.119,E2 17225.119} C_VEL
LIN {X 0,Y 488.977,Z 652.132,A -85,B 0,C 180,E1 17224.321,E2 17224.321} C_VEL
LIN {X 0,Y 487.506,Z 672.63,A -85,B 0,C 180,E1 17223.384,E2 17223.384} C_VEL
LIN {X 0,Y 485.759,Z 693.061,A -85,B 0,C 180,E1 17222.214,E2 17222.214} C_VEL
LIN {X 0,Y 483.895,Z 713.119,A -85,B 0,C 180,E1 17220.824,E2 17220.824} C_VEL
LIN {X 0,Y 482.014,Z 732.181,A -85,B 0,C 180,E1 17219.26,E2 17219.26} C_VEL
LIN {X 0,Y 480.419,Z 747.492,A -85,B 0,C 180,E1 17217.786,E2 17217.786} C_VEL
LIN {X 0,Y 478.521,Z 764.666,A -85,B 0,C 180,E1 17215.825,E2 17215.825} C_VEL
LIN {X 0,Y 476.946,Z 779.488,A -85,B 0,C 180,E1 17213.864,E2 17213.864} C_VEL
LIN {X 0,Y 475.467,Z 793.774,A -85,B 0,C 180,E1 17211.646,E2 17211.646} C_VEL
LIN {X 0,Y 474.28,Z 806.552,A -85,B 0,C 180,E1 17209.327,E2 17209.327} C_VEL
LIN {X 0,Y 473.36,Z 817.974,A -85,B 0,C 180,E1 17206.892,E2 17206.892} C_VEL
LIN {X 0,Y 472.718,Z 827.516,A -85,B 0,C 180,E1 17204.451,E2 17204.451} C_VEL
LIN {X 0,Y 472.305,Z 835.472,A -85,B 0,C 180,E1 17201.972,E2 17201.972} C_VEL
LIN {X 0,Y 472.075,Z 842.131,A -85,B 0,C 180,E1 17199.385,E2 17199.385} C_VEL
LIN {X 0,Y 471.958,Z 847.021,A -85,B 0,C 180,E1 17196.812,E2 17196.812} C_VEL
LIN {X 0,Y 471.914,Z 850.447,A -85,B 0,C 180,E1 17194.13,E2 17194.13} C_VEL
LIN {X 0,Y 471.898,Z 852.21,A -85,B 0,C 180,E1 17191.577,E2 17191.577} C_VEL
LIN {X 0,Y 471.909,Z 852.326,A -85,B 0,C 180,E1 17189.028,E2 17189.028} C_VEL
LIN {X 0,Y 471.909,Z 850.861,A -85,B 0,C 180,E1 17186.317,E2 17186.317} C_VEL
LIN {X 0,Y 471.94,Z 847.977,A -85,B 0,C 180,E1 17183.796,E2 17183.796} C_VEL
LIN {X 0,Y 472.02,Z 843.396,A -85,B 0,C 180,E1 17181.226,E2 17181.226} C_VEL
LIN {X 0,Y 472.233,Z 837.23,A -85,B 0,C 180,E1 17178.643,E2 17178.643} C_VEL
LIN {X 0,Y 472.6,Z 829.661,A -85,B 0,C 180,E1 17176.167,E2 17176.167} C_VEL
LIN {X 0,Y 473.217,Z 819.951,A -85,B 0,C 180,E1 17173.588,E2 17173.588} C_VEL
LIN {X 0,Y 474.075,Z 809.079,A -85,B 0,C 180,E1 17171.173,E2 17171.173} C_VEL
LIN {X 0,Y 475.154,Z 797.049,A -85,B 0,C 180,E1 17168.909,E2 17168.909} C_VEL
LIN {X 0,Y 476.475,Z 783.701,A -85,B 0,C 180,E1 17166.764,E2 17166.764} C_VEL
LIN {X 0,Y 478.089,Z 768.699,A -85,B 0,C 180,E1 17164.678,E2 17164.678} C_VEL
LIN {X 0,Y 479.924,Z 752.23,A -85,B 0,C 180,E1 17162.719,E2 17162.719} C_VEL
LIN {X 0,Y 481.558,Z 736.456,A -85,B 0,C 180,E1 17161.134,E2 17161.134} C_VEL
LIN {X 0,Y 483.423,Z 717.967,A -85,B 0,C 180,E1 17159.553,E2 17159.553} C_VEL
LIN {X 0,Y 485.197,Z 698.628,A -85,B 0,C 180,E1 17158.159,E2 17158.159} C_VEL
LIN {X 0,Y 486.915,Z 678.669,A -85,B 0,C 180,E1 17156.961,E2 17156.961} C_VEL
LIN {X 0,Y 488.5,Z 658.318,A -85,B 0,C 180,E1 17155.957,E2 17155.957} C_VEL
LIN {X 0,Y 489.826,Z 636.792,A -85,B 0,C 180,E1 17155.128,E2 17155.128} C_VEL
LIN {X 0,Y 490.935,Z 614.967,A -85,B 0,C 180,E1 17154.513,E2 17154.513} C_VEL
LIN {X 0,Y 491.649,Z 591.247,A -85,B 0,C 180,E1 17154.059,E2 17154.059} C_VEL
LIN {X 0,Y 495.438,Z 361.024,A -85,B 0,C 180,E1 17150.386,E2 17150.386} C_VEL
LIN {X 0,Y 495.87,Z 325.205,A -85,B 0,C 180,E1 17149.786,E2 17149.786} C_VEL
LIN {X 0,Y 492.327,Z 301.329,A -85,B 0,C 180,E1 17149.005,E2 17149.005} C_VEL
LIN {X 0,Y 492.462,Z 297.178,A -85,B 0,C 180,E1 17148.697,E2 17148.697} C_VEL
LIN {X 0,Y 482.324,Z 274.012,A -85,B 0,C 180,E1 17145.829,E2 17145.829} C_VEL
LIN {X 0,Y 474.603,Z 257.776,A -85,B 0,C 180,E1 17143.543,E2 17143.543} C_VEL
LIN {X 0,Y 472.975,Z 254.076,A -85,B 0,C 180,E1 17142.949,E2 17142.949} C_VEL
LIN {X 0,Y 472.95,Z 253.824,A -85,B 0,C 180,E1 17139.52,E2 17139.52} C_VEL
LIN {X 0,Y 472.949,Z 253.821,A -85,B 0,C 180,E1 17135.846,E2 17135.846} C_VEL
LIN {X 0,Y 472.945,Z 253.822,A -85,B 0,C 180,E1 17132.192,E2 17132.192} C_VEL
LIN {X 0,Y 472.942,Z 253.817,A -85,B 0,C 180,E1 17128.542,E2 17128.542} C_VEL
LIN {X 0,Y 472.951,Z 253.821,A -85,B 0,C 180,E1 17124.88,E2 17124.88} C_VEL
LIN {X 0,Y 472.939,Z 253.819,A -85,B 0,C 180,E1 17121.324,E2 17121.324} C_VEL
LIN {X 0,Y 472.941,Z 253.817,A -85,B 0,C 180,E1 17117.725,E2 17117.725} C_VEL
LIN {X 0,Y 472.955,Z 253.816,A -85,B 0,C 180,E1 17114.071,E2 17114.071} C_VEL
LIN {X 0,Y 472.95,Z 253.815,A -85,B 0,C 180,E1 17110.353,E2 17110.353} C_VEL
LIN {X 0,Y 472.95,Z 253.819,A -85,B 0,C 180,E1 17106.678,E2 17106.678} C_VEL
LIN {X 0,Y 472.924,Z 253.824,A -85,B 0,C 180,E1 17103.031,E2 17103.031} C_VEL
LIN {X 0,Y 472.918,Z 253.823,A -85,B 0,C 180,E1 17099.395,E2 17099.395} C_VEL
LIN {X 0,Y 472.943,Z 253.819,A -85,B 0,C 180,E1 17095.879,E2 17095.879} C_VEL
LIN {X 0,Y 472.958,Z 253.817,A -85,B 0,C 180,E1 17092.225,E2 17092.225} C_VEL
LIN {X 0,Y 472.921,Z 253.827,A -85,B 0,C 180,E1 17088.662,E2 17088.662} C_VEL
LIN {X 0,Y 472.9,Z 253.827,A -85,B 0,C 180,E1 17085.053,E2 17085.053} C_VEL
LIN {X 0,Y 472.913,Z 253.824,A -85,B 0,C 180,E1 17081.511,E2 17081.511} C_VEL
LIN {X 0,Y 472.962,Z 254.047,A -85,B 0,C 180,E1 17078.289,E2 17078.289} C_VEL
LIN {X 0,Y 475.855,Z 260.967,A -85,B 0,C 180,E1 17077.127,E2 17077.127} C_VEL
LIN {X 0,Y 481.513,Z 273.603,A -85,B 0,C 180,E1 17075.154,E2 17075.154} C_VEL
LIN {X 0,Y 489.025,Z 292.571,A -85,B 0,C 180,E1 17072.48,E2 17072.48} C_VEL
LIN {X 0,Y 488.667,Z 300.171,A -85,B 0,C 180,E1 17071.82,E2 17071.82} C_VEL
LIN {X 0,Y 492.924,Z 323.936,A -85,B 0,C 180,E1 17070.968,E2 17070.968} C_VEL
LIN {X 0,Y 487.894,Z 564.472,A -85,B 0,C 180,E1 17066.982,E2 17066.982} C_VEL
LIN {X 0,Y 487.582,Z 571.681,A -85,B 0,C 180,E1 17066.809,E2 17066.809} C_VEL
LIN {X 0,Y 485.85,Z 581.422,A -85,B 0,C 180,E1 17066.643,E2 17066.643} C_VEL
LIN {X 0,Y 480.247,Z 598.32,A -85,B 0,C 180,E1 17066.417,E2 17066.417} C_VEL
LIN {X 0,Y 479.033,Z 605.646,A -85,B 0,C 180,E1 17066.158,E2 17066.158} C_VEL
LIN {X 0,Y 477.509,Z 625.291,A -85,B 0,C 180,E1 17065.167,E2 17065.167} C_VEL
LIN {X 0,Y 475.747,Z 644.873,A -85,B 0,C 180,E1 17063.921,E2 17063.921} C_VEL
LIN {X 0,Y 473.978,Z 662.517,A -85,B 0,C 180,E1 17062.545,E2 17062.545} C_VEL
LIN {X 0,Y 472.211,Z 679.11,A -85,B 0,C 180,E1 17060.996,E2 17060.996} C_VEL
LIN {X 0,Y 470.384,Z 695.378,A -85,B 0,C 180,E1 17059.177,E2 17059.177} C_VEL
LIN {X 0,Y 468.722,Z 710.118,A -85,B 0,C 180,E1 17057.208,E2 17057.208} C_VEL
LIN {X 0,Y 467.312,Z 723.082,A -85,B 0,C 180,E1 17055.151,E2 17055.151} C_VEL
LIN {X 0,Y 466.146,Z 734.758,A -85,B 0,C 180,E1 17052.95,E2 17052.95} C_VEL
LIN {X 0,Y 465.227,Z 745.25,A -85,B 0,C 180,E1 17050.564,E2 17050.564} C_VEL
LIN {X 0,Y 464.606,Z 753.924,A -85,B 0,C 180,E1 17048.145,E2 17048.145} C_VEL
LIN {X 0,Y 464.233,Z 760.878,A -85,B 0,C 180,E1 17045.711,E2 17045.711} C_VEL
LIN {X 0,Y 464.024,Z 766.289,A -85,B 0,C 180,E1 17043.184,E2 17043.184} C_VEL
LIN {X 0,Y 463.951,Z 769.962,A -85,B 0,C 180,E1 17040.7,E2 17040.7} C_VEL
LIN {X 0,Y 463.922,Z 772.132,A -85,B 0,C 180,E1 17038.165,E2 17038.165} C_VEL
LIN {X 0,Y 463.914,Z 772.744,A -85,B 0,C 180,E1 17035.672,E2 17035.672} C_VEL
LIN {X 0,Y 463.925,Z 771.775,A -85,B 0,C 180,E1 17033.096,E2 17033.096} C_VEL
LIN {X 0,Y 463.951,Z 769.155,A -85,B 0,C 180,E1 17030.567,E2 17030.567} C_VEL
LIN {X 0,Y 464.06,Z 764.979,A -85,B 0,C 180,E1 17028.076,E2 17028.076} C_VEL
LIN {X 0,Y 464.311,Z 758.904,A -85,B 0,C 180,E1 17025.488,E2 17025.488} C_VEL
LIN {X 0,Y 464.773,Z 751.144,A -85,B 0,C 180,E1 17022.968,E2 17022.968} C_VEL
LIN {X 0,Y 465.446,Z 742.25,A -85,B 0,C 180,E1 17020.647,E2 17020.647} C_VEL
LIN {X 0,Y 466.394,Z 731.717,A -85,B 0,C 180,E1 17018.384,E2 17018.384} C_VEL
LIN {X 0,Y 467.647,Z 719.105,A -85,B 0,C 180,E1 17016.138,E2 17016.138} C_VEL
LIN {X 0,Y 469.058,Z 705.849,A -85,B 0,C 180,E1 17014.157,E2 17014.157} C_VEL
LIN {X 0,Y 470.706,Z 690.791,A -85,B 0,C 180,E1 17012.253,E2 17012.253} C_VEL
LIN {X 0,Y 472.531,Z 674.13,A -85,B 0,C 180,E1 17010.486,E2 17010.486} C_VEL
LIN {X 0,Y 474.321,Z 657.086,A -85,B 0,C 180,E1 17008.975,E2 17008.975} C_VEL
LIN {X 0,Y 476.034,Z 639.418,A -85,B 0,C 180,E1 17007.668,E2 17007.668} C_VEL
LIN {X 0,Y 477.683,Z 620.262,A -85,B 0,C 180,E1 17006.521,E2 17006.521} C_VEL
LIN {X 0,Y 479.043,Z 600.848,A -85,B 0,C 180,E1 17005.602,E2 17005.602} C_VEL
LIN {X 0,Y 480.215,Z 580.718,A -85,B 0,C 180,E1 17004.883,E2 17004.883} C_VEL
LIN {X 0,Y 481.052,Z 559.561,A -85,B 0,C 180,E1 17004.358,E2 17004.358} C_VEL
LIN {X 0,Y 485.902,Z 324.36,A -85,B 0,C 180,E1 17000.47,E2 17000.47} C_VEL
LIN {X 0,Y 481.369,Z 299.404,A -85,B 0,C 180,E1 16999.56,E2 16999.56} C_VEL
LIN {X 0,Y 481.504,Z 295.048,A -85,B 0,C 180,E1 16999.163,E2 16999.163} C_VEL
LIN {X 0,Y 474.324,Z 276.65,A -85,B 0,C 180,E1 16996.594,E2 16996.594} C_VEL
LIN {X 0,Y 467.803,Z 261.703,A -85,B 0,C 180,E1 16994.315,E2 16994.315} C_VEL
LIN {X 0,Y 465.022,Z 254.991,A -85,B 0,C 180,E1 16993.214,E2 16993.214} C_VEL
LIN {X 0,Y 465.009,Z 254.803,A -85,B 0,C 180,E1 16989.748,E2 16989.748} C_VEL
LIN {X 0,Y 465.007,Z 254.767,A -85,B 0,C 180,E1 16986.036,E2 16986.036} C_VEL
LIN {X 0,Y 465.013,Z 254.807,A -85,B 0,C 180,E1 16982.328,E2 16982.328} C_VEL
LIN {X 0,Y 465.008,Z 254.804,A -85,B 0,C 180,E1 16978.605,E2 16978.605} C_VEL
LIN {X 0,Y 464.994,Z 254.803,A -85,B 0,C 180,E1 16974.964,E2 16974.964} C_VEL
LIN {X 0,Y 465,Z 254.805,A -85,B 0,C 180,E1 16971.267,E2 16971.267} C_VEL
LIN {X 0,Y 465.012,Z 254.814,A -85,B 0,C 180,E1 16967.7,E2 16967.7} C_VEL
LIN {X 0,Y 465.012,Z 254.807,A -85,B 0,C 180,E1 16963.986,E2 16963.986} C_VEL
LIN {X 0,Y 465.005,Z 254.798,A -85,B 0,C 180,E1 16960.33,E2 16960.33} C_VEL
LIN {X 0,Y 464.991,Z 254.798,A -85,B 0,C 180,E1 16956.676,E2 16956.676} C_VEL
LIN {X 0,Y 464.997,Z 254.811,A -85,B 0,C 180,E1 16952.955,E2 16952.955} C_VEL
LIN {X 0,Y 465.013,Z 254.801,A -85,B 0,C 180,E1 16949.355,E2 16949.355} C_VEL
LIN {X 0,Y 465.011,Z 254.798,A -85,B 0,C 180,E1 16945.724,E2 16945.724} C_VEL
LIN {X 0,Y 465.003,Z 254.809,A -85,B 0,C 180,E1 16942.072,E2 16942.072} C_VEL
LIN {X 0,Y 464.989,Z 254.807,A -85,B 0,C 180,E1 16938.425,E2 16938.425} C_VEL
LIN {X 0,Y 465,Z 254.795,A -85,B 0,C 180,E1 16934.824,E2 16934.824} C_VEL
LIN {X 0,Y 465.012,Z 254.812,A -85,B 0,C 180,E1 16931.157,E2 16931.157} C_VEL
LIN {X 0,Y 465.013,Z 254.797,A -85,B 0,C 180,E1 16927.411,E2 16927.411} C_VEL
LIN {X 0,Y 465.002,Z 254.802,A -85,B 0,C 180,E1 16923.697,E2 16923.697} C_VEL
LIN {X 0,Y 464.986,Z 254.812,A -85,B 0,C 180,E1 16920.122,E2 16920.122} C_VEL
LIN {X 0,Y 464.992,Z 254.804,A -85,B 0,C 180,E1 16916.424,E2 16916.424} C_VEL
LIN {X 0,Y 465.017,Z 254.796,A -85,B 0,C 180,E1 16912.835,E2 16912.835} C_VEL
LIN {X 0,Y 465.013,Z 254.81,A -85,B 0,C 180,E1 16909.092,E2 16909.092} C_VEL
LIN {X 0,Y 465.008,Z 254.81,A -85,B 0,C 180,E1 16905.365,E2 16905.365} C_VEL
LIN {X 0,Y 464.987,Z 254.811,A -85,B 0,C 180,E1 16901.702,E2 16901.702} C_VEL
LIN {X 0,Y 464.987,Z 254.808,A -85,B 0,C 180,E1 16898.027,E2 16898.027} C_VEL
LIN {X 0,Y 465.006,Z 254.802,A -85,B 0,C 180,E1 16894.393,E2 16894.393} C_VEL
LIN {X 0,Y 465.016,Z 254.799,A -85,B 0,C 180,E1 16890.785,E2 16890.785} C_VEL
LIN {X 0,Y 464.997,Z 254.808,A -85,B 0,C 180,E1 16887.189,E2 16887.189} C_VEL
LIN {X 0,Y 464.982,Z 254.817,A -85,B 0,C 180,E1 16883.532,E2 16883.532} C_VEL
LIN {X 0,Y 464.988,Z 254.807,A -85,B 0,C 180,E1 16879.827,E2 16879.827} C_VEL
LIN {X 0,Y 465.017,Z 254.935,A -85,B 0,C 180,E1 16878.033,E2 16878.033} C_VEL
LIN {X 0,Y 465.427,Z 256.608,A -85,B 0,C 180,E1 16877.746,E2 16877.746} C_VEL
LIN {X 0,Y 467.464,Z 260.49,A -85,B 0,C 180,E1 16877.143,E2 16877.143} C_VEL
LIN {X 0,Y 474.987,Z 276.07,A -85,B 0,C 180,E1 16874.9,E2 16874.9} C_VEL
LIN {X 0,Y 483.315,Z 294.609,A -85,B 0,C 180,E1 16872.48,E2 16872.48} C_VEL
LIN {X 0,Y 486.126,Z 301.386,A -85,B 0,C 180,E1 16871.662,E2 16871.662} C_VEL
LIN {X 0,Y 489.994,Z 328.884,A -85,B 0,C 180,E1 16870.759,E2 16870.759} C_VEL
LIN {X 0,Y 485.91,Z 544.841,A -85,B 0,C 180,E1 16867.234,E2 16867.234} C_VEL
LIN {X 0,Y 484.653,Z 608.185,A -85,B 0,C 180,E1 16866.184,E2 16866.184} C_VEL
LIN {X 0,Y 483.587,Z 629.439,A -85,B 0,C 180,E1 16865.632,E2 16865.632} C_VEL
LIN {X 0,Y 482.163,Z 651.41,A -85,B 0,C 180,E1 16864.847,E2 16864.847} C_VEL
LIN {X 0,Y 480.547,Z 672.3,A -85,B 0,C 180,E1 16863.882,E2 16863.882} C_VEL
LIN {X 0,Y 478.77,Z 691.992,A -85,B 0,C 180,E1 16862.743,E2 16862.743} C_VEL
LIN {X 0,Y 476.754,Z 712.145,A -85,B 0,C 180,E1 16861.338,E2 16861.338} C_VEL
LIN {X 0,Y 474.811,Z 730.786,A -85,B 0,C 180,E1 16859.798,E2 16859.798} C_VEL
LIN {X 0,Y 472.841,Z 748.589,A -85,B 0,C 180,E1 16858.064,E2 16858.064} C_VEL
LIN {X 0,Y 471.029,Z 765.023,A -85,B 0,C 180,E1 16856.199,E2 16856.199} C_VEL
LIN {X 0,Y 469.596,Z 777.656,A -85,B 0,C 180,E1 16854.53,E2 16854.53} C_VEL
LIN {X 0,Y 467.99,Z 791.988,A -85,B 0,C 180,E1 16852.316,E2 16852.316} C_VEL
LIN {X 0,Y 466.637,Z 805.281,A -85,B 0,C 180,E1 16849.917,E2 16849.917} C_VEL
LIN {X 0,Y 465.624,Z 816.683,A -85,B 0,C 180,E1 16847.494,E2 16847.494} C_VEL
LIN {X 0,Y 464.866,Z 826.598,A -85,B 0,C 180,E1 16844.956,E2 16844.956} C_VEL
LIN {X 0,Y 464.365,Z 835.119,A -85,B 0,C 180,E1 16842.306,E2 16842.306} C_VEL
LIN {X 0,Y 464.094,Z 841.875,A -85,B 0,C 180,E1 16839.673,E2 16839.673} C_VEL
LIN {X 0,Y 463.971,Z 846.815,A -85,B 0,C 180,E1 16837.054,E2 16837.054} C_VEL
LIN {X 0,Y 463.918,Z 850.333,A -85,B 0,C 180,E1 16834.325,E2 16834.325} C_VEL
LIN {X 0,Y 463.903,Z 852.086,A -85,B 0,C 180,E1 16831.851,E2 16831.851} C_VEL
LIN {X 0,Y 463.901,Z 852.371,A -85,B 0,C 180,E1 16829.258,E2 16829.258} C_VEL
LIN {X 0,Y 463.914,Z 851.234,A -85,B 0,C 180,E1 16826.663,E2 16826.663} C_VEL
LIN {X 0,Y 463.938,Z 848.455,A -85,B 0,C 180,E1 16824.061,E2 16824.061} C_VEL
LIN {X 0,Y 464.021,Z 843.904,A -85,B 0,C 180,E1 16821.324,E2 16821.324} C_VEL
LIN {X 0,Y 464.225,Z 838.246,A -85,B 0,C 180,E1 16818.822,E2 16818.822} C_VEL
LIN {X 0,Y 464.595,Z 830.876,A -85,B 0,C 180,E1 16816.305,E2 16816.305} C_VEL
LIN {X 0,Y 465.247,Z 821.345,A -85,B 0,C 180,E1 16813.647,E2 16813.647} C_VEL
LIN {X 0,Y 466.182,Z 810.345,A -85,B 0,C 180,E1 16811.102,E2 16811.102} C_VEL
LIN {X 0,Y 467.388,Z 797.748,A -85,B 0,C 180,E1 16808.673,E2 16808.673} C_VEL
LIN {X 0,Y 468.903,Z 783.699,A -85,B 0,C 180,E1 16806.366,E2 16806.366} C_VEL
LIN {X 0,Y 470.623,Z 768.795,A -85,B 0,C 180,E1 16804.265,E2 16804.265} C_VEL
LIN {X 0,Y 472.387,Z 752.699,A -85,B 0,C 180,E1 16802.383,E2 16802.383} C_VEL
LIN {X 0,Y 474.306,Z 734.71,A -85,B 0,C 180,E1 16800.581,E2 16800.581} C_VEL
LIN {X 0,Y 476.31,Z 715.986,A -85,B 0,C 180,E1 16798.978,E2 16798.978} C_VEL
LIN {X 0,Y 478.208,Z 696.74,A -85,B 0,C 180,E1 16797.585,E2 16797.585} C_VEL
LIN {X 0,Y 480.019,Z 676.885,A -85,B 0,C 180,E1 16796.398,E2 16796.398} C_VEL
LIN {X 0,Y 481.7,Z 655.938,A -85,B 0,C 180,E1 16795.373,E2 16795.373} C_VEL
LIN {X 0,Y 483.143,Z 634.52,A -85,B 0,C 180,E1 16794.555,E2 16794.555} C_VEL
LIN {X 0,Y 484.246,Z 613.355,A -85,B 0,C 180,E1 16793.969,E2 16793.969} C_VEL
LIN {X 0,Y 485.014,Z 586.377,A -85,B 0,C 180,E1 16793.467,E2 16793.467} C_VEL
LIN {X 0,Y 489.037,Z 360.053,A -85,B 0,C 180,E1 16789.81,E2 16789.81} C_VEL
LIN {X 0,Y 489.486,Z 326.59,A -85,B 0,C 180,E1 16789.24,E2 16789.24} C_VEL
LIN {X 0,Y 485.796,Z 301.395,A -85,B 0,C 180,E1 16788.403,E2 16788.403} C_VEL
LIN {X 0,Y 478.4,Z 283.662,A -85,B 0,C 180,E1 16786.227,E2 16786.227} C_VEL
LIN {X 0,Y 470.837,Z 267.222,A -85,B 0,C 180,E1 16783.953,E2 16783.953} C_VEL
LIN {X 0,Y 466.528,Z 258.607,A -85,B 0,C 180,E1 16782.629,E2 16782.629} C_VEL
LIN {X 0,Y 465.049,Z 255.099,A -85,B 0,C 180,E1 16782.055,E2 16782.055} C_VEL
LIN {X 0,Y 464.995,Z 254.811,A -85,B 0,C 180,E1 16780.495,E2 16780.495} C_VEL
LIN {X 0,Y 465.004,Z 254.813,A -85,B 0,C 180,E1 16776.864,E2 16776.864} C_VEL
LIN {X 0,Y 465.011,Z 254.812,A -85,B 0,C 180,E1 16773.235,E2 16773.235} C_VEL
LIN {X 0,Y 465.006,Z 254.806,A -85,B 0,C 180,E1 16769.499,E2 16769.499} C_VEL
LIN {X 0,Y 465.008,Z 254.808,A -85,B 0,C 180,E1 16765.881,E2 16765.881} C_VEL
LIN {X 0,Y 465.009,Z 254.812,A -85,B 0,C 180,E1 16762.237,E2 16762.237} C_VEL
LIN {X 0,Y 465.011,Z 254.812,A -85,B 0,C 180,E1 16758.515,E2 16758.515} C_VEL
LIN {X 0,Y 465.011,Z 254.807,A -85,B 0,C 180,E1 16754.826,E2 16754.826} C_VEL
LIN {X 0,Y 464.992,Z 254.803,A -85,B 0,C 180,E1 16751.159,E2 16751.159} C_VEL
LIN {X 0,Y 464.987,Z 254.808,A -85,B 0,C 180,E1 16747.414,E2 16747.414} C_VEL
LIN {X 0,Y 465.001,Z 254.809,A -85,B 0,C 180,E1 16743.823,E2 16743.823} C_VEL
LIN {X 0,Y 465.018,Z 254.811,A -85,B 0,C 180,E1 16740.124,E2 16740.124} C_VEL
LIN {X 0,Y 465.008,Z 254.813,A -85,B 0,C 180,E1 16736.426,E2 16736.426} C_VEL
LIN {X 0,Y 464.977,Z 254.808,A -85,B 0,C 180,E1 16732.837,E2 16732.837} C_VEL
LIN {X 0,Y 464.969,Z 254.818,A -85,B 0,C 180,E1 16729.219,E2 16729.219} C_VEL
LIN {X 0,Y 464.988,Z 254.811,A -85,B 0,C 180,E1 16725.684,E2 16725.684} C_VEL
LIN {X 0,Y 465.01,Z 254.812,A -85,B 0,C 180,E1 16722.094,E2 16722.094} C_VEL
LIN {X 0,Y 464.986,Z 255.002,A -85,B 0,C 180,E1 16719.22,E2 16719.22} C_VEL
LIN {X 0,Y 466.235,Z 258.243,A -85,B 0,C 180,E1 16718.62,E2 16718.62} C_VEL
LIN {X 0,Y 470.727,Z 267.911,A -85,B 0,C 180,E1 16716.995,E2 16716.995} C_VEL
LIN {X 0,Y 477.735,Z 284.377,A -85,B 0,C 180,E1 16714.462,E2 16714.462} C_VEL
LIN {X 0,Y 482.31,Z 296.415,A -85,B 0,C 180,E1 16712.77,E2 16712.77} C_VEL
LIN {X 0,Y 482.163,Z 300.405,A -85,B 0,C 180,E1 16712.449,E2 16712.449} C_VEL
LIN {X 0,Y 486.624,Z 325.454,A -85,B 0,C 180,E1 16711.528,E2 16711.528} C_VEL
LIN {X 0,Y 481.215,Z 564.929,A -85,B 0,C 180,E1 16707.5,E2 16707.5} C_VEL
LIN {X 0,Y 480.248,Z 585.877,A -85,B 0,C 180,E1 16706.925,E2 16706.925} C_VEL
LIN {X 0,Y 479.033,Z 605.646,A -85,B 0,C 180,E1 16706.158,E2 16706.158} C_VEL
LIN {X 0,Y 477.683,Z 612.988,A -85,B 0,C 180,E1 16705.885,E2 16705.885} C_VEL
LIN {X 0,Y 471.025,Z 631.404,A -85,B 0,C 180,E1 16705.278,E2 16705.278} C_VEL
LIN {X 0,Y 469.511,Z 638.19,A -85,B 0,C 180,E1 16704.907,E2 16704.907} C_VEL
LIN {X 0,Y 467.669,Z 655.968,A -85,B 0,C 180,E1 16703.606,E2 16703.606} C_VEL
LIN {X 0,Y 465.751,Z 673.079,A -85,B 0,C 180,E1 16702.098,E2 16702.098} C_VEL
LIN {X 0,Y 463.856,Z 689.223,A -85,B 0,C 180,E1 16700.4,E2 16700.4} C_VEL
LIN {X 0,Y 462.017,Z 704.518,A -85,B 0,C 180,E1 16698.486,E2 16698.486} C_VEL
LIN {X 0,Y 460.283,Z 719.046,A -85,B 0,C 180,E1 16696.31,E2 16696.31} C_VEL
LIN {X 0,Y 458.859,Z 731.742,A -85,B 0,C 180,E1 16694.024,E2 16694.024} C_VEL
LIN {X 0,Y 457.793,Z 742.152,A -85,B 0,C 180,E1 16691.771,E2 16691.771} C_VEL
LIN {X 0,Y 457.003,Z 751.287,A -85,B 0,C 180,E1 16689.383,E2 16689.383} C_VEL
LIN {X 0,Y 456.466,Z 758.988,A -85,B 0,C 180,E1 16686.884,E2 16686.884} C_VEL
LIN {X 0,Y 456.169,Z 764.872,A -85,B 0,C 180,E1 16684.438,E2 16684.438} C_VEL
LIN {X 0,Y 456.022,Z 769.285,A -85,B 0,C 180,E1 16681.899,E2 16681.899} C_VEL
LIN {X 0,Y 455.962,Z 772.035,A -85,B 0,C 180,E1 16679.421,E2 16679.421} C_VEL
LIN {X 0,Y 455.951,Z 773.366,A -85,B 0,C 180,E1 16676.813,E2 16676.813} C_VEL
LIN {X 0,Y 455.955,Z 773.101,A -85,B 0,C 180,E1 16674.21,E2 16674.21} C_VEL
LIN {X 0,Y 455.967,Z 771.235,A -85,B 0,C 180,E1 16671.608,E2 16671.608} C_VEL
LIN {X 0,Y 456.054,Z 767.756,A -85,B 0,C 180,E1 16669.068,E2 16669.068} C_VEL
LIN {X 0,Y 456.244,Z 762.72,A -85,B 0,C 180,E1 16666.554,E2 16666.554} C_VEL
LIN {X 0,Y 456.648,Z 755.703,A -85,B 0,C 180,E1 16663.938,E2 16663.938} C_VEL
LIN {X 0,Y 457.278,Z 747.3,A -85,B 0,C 180,E1 16661.478,E2 16661.478} C_VEL
LIN {X 0,Y 458.17,Z 737.64,A -85,B 0,C 180,E1 16659.168,E2 16659.168} C_VEL
LIN {X 0,Y 459.374,Z 726.065,A -85,B 0,C 180,E1 16656.877,E2 16656.877} C_VEL
LIN {X 0,Y 460.834,Z 713.052,A -85,B 0,C 180,E1 16654.731,E2 16654.731} C_VEL
LIN {X 0,Y 462.465,Z 699.076,A -85,B 0,C 180,E1 16652.785,E2 16652.785} C_VEL
LIN {X 0,Y 464.319,Z 683.274,A -85,B 0,C 180,E1 16650.927,E2 16650.927} C_VEL
LIN {X 0,Y 466.262,Z 666.387,A -85,B 0,C 180,E1 16649.264,E2 16649.264} C_VEL
LIN {X 0,Y 468.097,Z 649.355,A -85,B 0,C 180,E1 16647.859,E2 16647.859} C_VEL
LIN {X 0,Y 469.942,Z 630.561,A -85,B 0,C 180,E1 16646.586,E2 16646.586} C_VEL
LIN {X 0,Y 471.506,Z 611.67,A -85,B 0,C 180,E1 16645.562,E2 16645.562} C_VEL
LIN {X 0,Y 472.869,Z 591.836,A -85,B 0,C 180,E1 16644.724,E2 16644.724} C_VEL
LIN {X 0,Y 473.975,Z 570.504,A -85,B 0,C 180,E1 16644.068,E2 16644.068} C_VEL
LIN {X 0,Y 474.721,Z 546.308,A -85,B 0,C 180,E1 16643.59,E2 16643.59} C_VEL
LIN {X 0,Y 479.523,Z 325.678,A -85,B 0,C 180,E1 16639.905,E2 16639.905} C_VEL
LIN {X 0,Y 474.791,Z 299.167,A -85,B 0,C 180,E1 16638.905,E2 16638.905} C_VEL
LIN {X 0,Y 469.24,Z 284.328,A -85,B 0,C 180,E1 16636.841,E2 16636.841} C_VEL
LIN {X 0,Y 462.195,Z 267.533,A -85,B 0,C 180,E1 16634.287,E2 16634.287} C_VEL
LIN {X 0,Y 457.13,Z 256.176,A -85,B 0,C 180,E1 16632.401,E2 16632.401} C_VEL
LIN {X 0,Y 457.066,Z 255.756,A -85,B 0,C 180,E1 16631.904,E2 16631.904} C_VEL
LIN {X 0,Y 457.069,Z 255.781,A -85,B 0,C 180,E1 16628.17,E2 16628.17} C_VEL
LIN {X 0,Y 457.071,Z 255.783,A -85,B 0,C 180,E1 16624.474,E2 16624.474} C_VEL
LIN {X 0,Y 457.063,Z 255.798,A -85,B 0,C 180,E1 16620.787,E2 16620.787} C_VEL
LIN {X 0,Y 457.056,Z 255.799,A -85,B 0,C 180,E1 16617.141,E2 16617.141} C_VEL
LIN {X 0,Y 457.064,Z 255.794,A -85,B 0,C 180,E1 16613.399,E2 16613.399} C_VEL
LIN {X 0,Y 457.074,Z 255.787,A -85,B 0,C 180,E1 16609.766,E2 16609.766} C_VEL
LIN {X 0,Y 457.072,Z 255.787,A -85,B 0,C 180,E1 16606.027,E2 16606.027} C_VEL
LIN {X 0,Y 457.07,Z 255.795,A -85,B 0,C 180,E1 16602.323,E2 16602.323} C_VEL
LIN {X 0,Y 457.053,Z 255.8,A -85,B 0,C 180,E1 16598.653,E2 16598.653} C_VEL
LIN {X 0,Y 457.056,Z 255.793,A -85,B 0,C 180,E1 16594.883,E2 16594.883} C_VEL
LIN {X 0,Y 457.072,Z 255.784,A -85,B 0,C 180,E1 16591.208,E2 16591.208} C_VEL
LIN {X 0,Y 457.076,Z 255.801,A -85,B 0,C 180,E1 16587.486,E2 16587.486} C_VEL
LIN {X 0,Y 457.074,Z 255.791,A -85,B 0,C 180,E1 16583.733,E2 16583.733} C_VEL
LIN {X 0,Y 457.059,Z 255.785,A -85,B 0,C 180,E1 16580.086,E2 16580.086} C_VEL
LIN {X 0,Y 457.049,Z 255.799,A -85,B 0,C 180,E1 16576.391,E2 16576.391} C_VEL
LIN {X 0,Y 457.057,Z 255.792,A -85,B 0,C 180,E1 16572.673,E2 16572.673} C_VEL
LIN {X 0,Y 457.07,Z 255.784,A -85,B 0,C 180,E1 16568.934,E2 16568.934} C_VEL
LIN {X 0,Y 457.074,Z 255.8,A -85,B 0,C 180,E1 16565.27,E2 16565.27} C_VEL
LIN {X 0,Y 457.073,Z 255.79,A -85,B 0,C 180,E1 16561.486,E2 16561.486} C_VEL
LIN {X 0,Y 457.05,Z 255.784,A -85,B 0,C 180,E1 16557.868,E2 16557.868} C_VEL
LIN {X 0,Y 457.049,Z 255.797,A -85,B 0,C 180,E1 16554.224,E2 16554.224} C_VEL
LIN {X 0,Y 457.065,Z 255.8,A -85,B 0,C 180,E1 16550.556,E2 16550.556} C_VEL
LIN {X 0,Y 457.075,Z 255.785,A -85,B 0,C 180,E1 16546.849,E2 16546.849} C_VEL
LIN {X 0,Y 457.071,Z 255.786,A -85,B 0,C 180,E1 16543.216,E2 16543.216} C_VEL
LIN {X 0,Y 457.052,Z 255.794,A -85,B 0,C 180,E1 16539.511,E2 16539.511} C_VEL
LIN {X 0,Y 457.046,Z 255.796,A -85,B 0,C 180,E1 16535.814,E2 16535.814} C_VEL
LIN {X 0,Y 457.055,Z 255.794,A -85,B 0,C 180,E1 16532.085,E2 16532.085} C_VEL
LIN {X 0,Y 457.077,Z 255.792,A -85,B 0,C 180,E1 16528.478,E2 16528.478} C_VEL
LIN {X 0,Y 457.075,Z 255.79,A -85,B 0,C 180,E1 16524.724,E2 16524.724} C_VEL
LIN {X 0,Y 457.056,Z 255.8,A -85,B 0,C 180,E1 16521.108,E2 16521.108} C_VEL
LIN {X 0,Y 457.103,Z 256.04,A -85,B 0,C 180,E1 16518.905,E2 16518.905} C_VEL
LIN {X 0,Y 458.601,Z 259.596,A -85,B 0,C 180,E1 16518.319,E2 16518.319} C_VEL
LIN {X 0,Y 465.492,Z 273.557,A -85,B 0,C 180,E1 16516.194,E2 16516.194} C_VEL
LIN {X 0,Y 474.121,Z 292.386,A -85,B 0,C 180,E1 16513.596,E2 16513.596} C_VEL
LIN {X 0,Y 478.502,Z 302.419,A -85,B 0,C 180,E1 16512.36,E2 16512.36} C_VEL
LIN {X 0,Y 480.208,Z 305.761,A -85,B 0,C 180,E1 16512.122,E2 16512.122} C_VEL
LIN {X 0,Y 483.689,Z 330.294,A -85,B 0,C 180,E1 16511.324,E2 16511.324} C_VEL
LIN {X 0,Y 479.316,Z 546.111,A -85,B 0,C 180,E1 16507.758,E2 16507.758} C_VEL
LIN {X 0,Y 478.002,Z 607.802,A -85,B 0,C 180,E1 16506.723,E2 16506.723} C_VEL
LIN {X 0,Y 476.872,Z 629.112,A -85,B 0,C 180,E1 16506.165,E2 16506.165} C_VEL
LIN {X 0,Y 475.372,Z 650.986,A -85,B 0,C 180,E1 16505.374,E2 16505.374} C_VEL
LIN {X 0,Y 473.719,Z 671.029,A -85,B 0,C 180,E1 16504.446,E2 16504.446} C_VEL
LIN {X 0,Y 471.819,Z 690.917,A -85,B 0,C 180,E1 16503.287,E2 16503.287} C_VEL
LIN {X 0,Y 469.627,Z 711.465,A -85,B 0,C 180,E1 16501.843,E2 16501.843} C_VEL
LIN {X 0,Y 467.58,Z 729.881,A -85,B 0,C 180,E1 16500.307,E2 16500.307} C_VEL
LIN {X 0,Y 465.444,Z 747.943,A -85,B 0,C 180,E1 16498.525,E2 16498.525} C_VEL
LIN {X 0,Y 463.47,Z 764.711,A -85,B 0,C 180,E1 16496.591,E2 16496.591} C_VEL
LIN {X 0,Y 461.716,Z 779.978,A -85,B 0,C 180,E1 16494.56,E2 16494.56} C_VEL
LIN {X 0,Y 460.295,Z 792.596,A -85,B 0,C 180,E1 16492.603,E2 16492.603} C_VEL
LIN {X 0,Y 458.789,Z 806.267,A -85,B 0,C 180,E1 16490.066,E2 16490.066} C_VEL
LIN {X 0,Y 457.744,Z 817.235,A -85,B 0,C 180,E1 16487.674,E2 16487.674} C_VEL
LIN {X 0,Y 456.932,Z 827.056,A -85,B 0,C 180,E1 16485.092,E2 16485.092} C_VEL
LIN {X 0,Y 456.394,Z 835.472,A -85,B 0,C 180,E1 16482.396,E2 16482.396} C_VEL
LIN {X 0,Y 456.103,Z 842.131,A -85,B 0,C 180,E1 16479.716,E2 16479.716} C_VEL
LIN {X 0,Y 455.979,Z 846.815,A -85,B 0,C 180,E1 16477.179,E2 16477.179} C_VEL
LIN {X 0,Y 455.92,Z 850.333,A -85,B 0,C 180,E1 16474.401,E2 16474.401} C_VEL
LIN {X 0,Y 455.903,Z 852.086,A -85,B 0,C 180,E1 16471.884,E2 16471.884} C_VEL
LIN {X 0,Y 455.901,Z 852.371,A -85,B 0,C 180,E1 16469.245,E2 16469.245} C_VEL
LIN {X 0,Y 455.913,Z 851.234,A -85,B 0,C 180,E1 16466.604,E2 16466.604} C_VEL
LIN {X 0,Y 455.938,Z 848.615,A -85,B 0,C 180,E1 16464.083,E2 16464.083} C_VEL
LIN {X 0,Y 456.025,Z 844.412,A -85,B 0,C 180,E1 16461.424,E2 16461.424} C_VEL
LIN {X 0,Y 456.228,Z 838.853,A -85,B 0,C 180,E1 16458.879,E2 16458.879} C_VEL
LIN {X 0,Y 456.641,Z 831.281,A -85,B 0,C 180,E1 16456.191,E2 16456.191} C_VEL
LIN {X 0,Y 457.302,Z 822.373,A -85,B 0,C 180,E1 16453.616,E2 16453.616} C_VEL
LIN {X 0,Y 458.216,Z 812.084,A -85,B 0,C 180,E1 16451.158,E2 16451.158} C_VEL
LIN {X 0,Y 459.471,Z 799.849,A -85,B 0,C 180,E1 16448.689,E2 16448.689} C_VEL
LIN {X 0,Y 460.857,Z 787.744,A -85,B 0,C 180,E1 16446.596,E2 16446.596} C_VEL
LIN {X 0,Y 462.58,Z 772.244,A -85,B 0,C 180,E1 16444.385,E2 16444.385} C_VEL
LIN {X 0,Y 464.478,Z 755.75,A -85,B 0,C 180,E1 16442.36,E2 16442.36} C_VEL
LIN {X 0,Y 466.489,Z 738.504,A -85,B 0,C 180,E1 16440.533,E2 16440.533} C_VEL
LIN {X 0,Y 468.548,Z 720.434,A -85,B 0,C 180,E1 16438.907,E2 16438.907} C_VEL
LIN {X 0,Y 470.635,Z 700.802,A -85,B 0,C 180,E1 16437.408,E2 16437.408} C_VEL
LIN {X 0,Y 472.667,Z 680.606,A -85,B 0,C 180,E1 16436.123,E2 16436.123} C_VEL
LIN {X 0,Y 474.439,Z 660.654,A -85,B 0,C 180,E1 16435.09,E2 16435.09} C_VEL
LIN {X 0,Y 476.008,Z 639.044,A -85,B 0,C 180,E1 16434.204,E2 16434.204} C_VEL
LIN {X 0,Y 477.354,Z 616.867,A -85,B 0,C 180,E1 16433.532,E2 16433.532} C_VEL
LIN {X 0,Y 478.204,Z 594.619,A -85,B 0,C 180,E1 16433.072,E2 16433.072} C_VEL
LIN {X 0,Y 482.559,Z 365.528,A -85,B 0,C 180,E1 16429.326,E2 16429.326} C_VEL
LIN {X 0,Y 483.154,Z 327.999,A -85,B 0,C 180,E1 16428.679,E2 16428.679} C_VEL
LIN {X 0,Y 479.527,Z 304.478,A -85,B 0,C 180,E1 16427.883,E2 16427.883} C_VEL
LIN {X 0,Y 477.764,Z 301.384,A -85,B 0,C 180,E1 16427.626,E2 16427.626} C_VEL
LIN {X 0,Y 469.764,Z 282.74,A -85,B 0,C 180,E1 16425.209,E2 16425.209} C_VEL
LIN {X 0,Y 462.824,Z 268.005,A -85,B 0,C 180,E1 16423.053,E2 16423.053} C_VEL
LIN {X 0,Y 458.551,Z 259.519,A -85,B 0,C 180,E1 16421.686,E2 16421.686} C_VEL
LIN {X 0,Y 457.115,Z 256.089,A -85,B 0,C 180,E1 16421.094,E2 16421.094} C_VEL
LIN {X 0,Y 457.074,Z 255.802,A -85,B 0,C 180,E1 16419.051,E2 16419.051} C_VEL
LIN {X 0,Y 457.072,Z 255.802,A -85,B 0,C 180,E1 16415.276,E2 16415.276} C_VEL
LIN {X 0,Y 457.068,Z 255.796,A -85,B 0,C 180,E1 16411.522,E2 16411.522} C_VEL
LIN {X 0,Y 457.072,Z 255.803,A -85,B 0,C 180,E1 16407.772,E2 16407.772} C_VEL
LIN {X 0,Y 457.072,Z 255.795,A -85,B 0,C 180,E1 16404.01,E2 16404.01} C_VEL
LIN {X 0,Y 457.07,Z 255.793,A -85,B 0,C 180,E1 16400.355,E2 16400.355} C_VEL
LIN {X 0,Y 457.074,Z 255.795,A -85,B 0,C 180,E1 16396.636,E2 16396.636} C_VEL
LIN {X 0,Y 457.061,Z 255.8,A -85,B 0,C 180,E1 16393.023,E2 16393.023} C_VEL
LIN {X 0,Y 457.05,Z 255.803,A -85,B 0,C 180,E1 16389.317,E2 16389.317} C_VEL
LIN {X 0,Y 457.056,Z 255.8,A -85,B 0,C 180,E1 16385.65,E2 16385.65} C_VEL
LIN {X 0,Y 457.073,Z 255.795,A -85,B 0,C 180,E1 16382.007,E2 16382.007} C_VEL
LIN {X 0,Y 457.074,Z 255.793,A -85,B 0,C 180,E1 16378.371,E2 16378.371} C_VEL
LIN {X 0,Y 457.048,Z 255.801,A -85,B 0,C 180,E1 16374.729,E2 16374.729} C_VEL
LIN {X 0,Y 457.032,Z 255.805,A -85,B 0,C 180,E1 16371.192,E2 16371.192} C_VEL
LIN {X 0,Y 457.037,Z 255.801,A -85,B 0,C 180,E1 16367.493,E2 16367.493} C_VEL
LIN {X 0,Y 457.075,Z 255.799,A -85,B 0,C 180,E1 16364.002,E2 16364.002} C_VEL
LIN {X 0,Y 457.067,Z 255.853,A -85,B 0,C 180,E1 16360.248,E2 16360.248} C_VEL
LIN {X 0,Y 457.375,Z 257.213,A -85,B 0,C 180,E1 16359.929,E2 16359.929} C_VEL
LIN {X 0,Y 462.74,Z 268.535,A -85,B 0,C 180,E1 16357.917,E2 16357.917} C_VEL
LIN {X 0,Y 469.668,Z 284.573,A -85,B 0,C 180,E1 16355.34,E2 16355.34} C_VEL
LIN {X 0,Y 475.628,Z 299.915,A -85,B 0,C 180,E1 16353.131,E2 16353.131} C_VEL
LIN {X 0,Y 480.373,Z 326.936,A -85,B 0,C 180,E1 16352.104,E2 16352.104} C_VEL
LIN {X 0,Y 474.577,Z 565.413,A -85,B 0,C 180,E1 16348.032,E2 16348.032} C_VEL
LIN {X 0,Y 473.557,Z 586.286,A -85,B 0,C 180,E1 16347.452,E2 16347.452} C_VEL
LIN {X 0,Y 472.271,Z 606.066,A -85,B 0,C 180,E1 16346.676,E2 16346.676} C_VEL
LIN {X 0,Y 470.662,Z 625.714,A -85,B 0,C 180,E1 16345.676,E2 16345.676} C_VEL
LIN {X 0,Y 469.511,Z 638.19,A -85,B 0,C 180,E1 16344.907,E2 16344.907} C_VEL
LIN {X 0,Y 467.967,Z 645.078,A -85,B 0,C 180,E1 16344.505,E2 16344.505} C_VEL
LIN {X 0,Y 460.861,Z 662.344,A -85,B 0,C 180,E1 16343.55,E2 16343.55} C_VEL
LIN {X 0,Y 459.254,Z 668.616,A -85,B 0,C 180,E1 16343.048,E2 16343.048} C_VEL
LIN {X 0,Y 457.207,Z 684.922,A -85,B 0,C 180,E1 16341.396,E2 16341.396} C_VEL
LIN {X 0,Y 455.158,Z 700.859,A -85,B 0,C 180,E1 16339.471,E2 16339.471} C_VEL
LIN {X 0,Y 453.35,Z 714.951,A -85,B 0,C 180,E1 16337.447,E2 16337.447} C_VEL
LIN {X 0,Y 451.774,Z 727.723,A -85,B 0,C 180,E1 16335.27,E2 16335.27} C_VEL
LIN {X 0,Y 450.454,Z 739.302,A -85,B 0,C 180,E1 16332.907,E2 16332.907} C_VEL
LIN {X 0,Y 449.413,Z 749.562,A -85,B 0,C 180,E1 16330.349,E2 16330.349} C_VEL
LIN {X 0,Y 448.727,Z 757.786,A -85,B 0,C 180,E1 16327.79,E2 16327.79} C_VEL
LIN {X 0,Y 448.318,Z 764.099,A -85,B 0,C 180,E1 16325.285,E2 16325.285} C_VEL
LIN {X 0,Y 448.103,Z 768.985,A -85,B 0,C 180,E1 16322.683,E2 16322.683} C_VEL
LIN {X 0,Y 448.011,Z 772.207,A -85,B 0,C 180,E1 16320.143,E2 16320.143} C_VEL
LIN {X 0,Y 447.985,Z 773.943,A -85,B 0,C 180,E1 16317.518,E2 16317.518} C_VEL
LIN {X 0,Y 447.982,Z 774.054,A -85,B 0,C 180,E1 16314.952,E2 16314.952} C_VEL
LIN {X 0,Y 448.006,Z 772.609,A -85,B 0,C 180,E1 16312.298,E2 16312.298} C_VEL
LIN {X 0,Y 448.068,Z 769.575,A -85,B 0,C 180,E1 16309.669,E2 16309.669} C_VEL
LIN {X 0,Y 448.256,Z 765.083,A -85,B 0,C 180,E1 16307.125,E2 16307.125} C_VEL
LIN {X 0,Y 448.634,Z 758.568,A -85,B 0,C 180,E1 16304.456,E2 16304.456} C_VEL
LIN {X 0,Y 449.244,Z 750.634,A -85,B 0,C 180,E1 16301.947,E2 16301.947} C_VEL
LIN {X 0,Y 450.133,Z 741.195,A -85,B 0,C 180,E1 16299.529,E2 16299.529} C_VEL
LIN {X 0,Y 451.388,Z 729.708,A -85,B 0,C 180,E1 16297.106,E2 16297.106} C_VEL
LIN {X 0,Y 452.957,Z 716.608,A -85,B 0,C 180,E1 16294.813,E2 16294.813} C_VEL
LIN {X 0,Y 454.697,Z 702.741,A -85,B 0,C 180,E1 16292.774,E2 16292.774} C_VEL
LIN {X 0,Y 456.645,Z 687.464,A -85,B 0,C 180,E1 16290.88,E2 16290.88} C_VEL
LIN {X 0,Y 458.733,Z 670.554,A -85,B 0,C 180,E1 16289.127,E2 16289.127} C_VEL
LIN {X 0,Y 460.698,Z 653.276,A -85,B 0,C 180,E1 16287.638,E2 16287.638} C_VEL
LIN {X 0,Y 462.621,Z 635.129,A -85,B 0,C 180,E1 16286.346,E2 16286.346} C_VEL
LIN {X 0,Y 464.363,Z 616.123,A -85,B 0,C 180,E1 16285.246,E2 16285.246} C_VEL
LIN {X 0,Y 465.888,Z 596.313,A -85,B 0,C 180,E1 16284.347,E2 16284.347} C_VEL
LIN {X 0,Y 467.104,Z 575.997,A -85,B 0,C 180,E1 16283.661,E2 16283.661} C_VEL
LIN {X 0,Y 467.929,Z 554.304,A -85,B 0,C 180,E1 16283.175,E2 16283.175} C_VEL
LIN {X 0,Y 473.223,Z 327.187,A -85,B 0,C 180,E1 16279.332,E2 16279.332} C_VEL
LIN {X 0,Y 468.524,Z 302.339,A -85,B 0,C 180,E1 16278.378,E2 16278.378} C_VEL
LIN {X 0,Y 466.918,Z 299.276,A -85,B 0,C 180,E1 16278.121,E2 16278.121} C_VEL
LIN {X 0,Y 459.107,Z 279.566,A -85,B 0,C 180,E1 16275.223,E2 16275.223} C_VEL
LIN {X 0,Y 452.313,Z 264.289,A -85,B 0,C 180,E1 16272.731,E2 16272.731} C_VEL
LIN {X 0,Y 449.178,Z 257.148,A -85,B 0,C 180,E1 16271.483,E2 16271.483} C_VEL
LIN {X 0,Y 449.122,Z 256.748,A -85,B 0,C 180,E1 16270.899,E2 16270.899} C_VEL
LIN {X 0,Y 449.113,Z 256.747,A -85,B 0,C 180,E1 16267.21,E2 16267.21} C_VEL
LIN {X 0,Y 449.125,Z 256.794,A -85,B 0,C 180,E1 16263.42,E2 16263.42} C_VEL
LIN {X 0,Y 449.138,Z 256.791,A -85,B 0,C 180,E1 16259.648,E2 16259.648} C_VEL
LIN {X 0,Y 449.134,Z 256.791,A -85,B 0,C 180,E1 16255.877,E2 16255.877} C_VEL
LIN {X 0,Y 449.137,Z 256.789,A -85,B 0,C 180,E1 16252.092,E2 16252.092} C_VEL
LIN {X 0,Y 449.136,Z 256.787,A -85,B 0,C 180,E1 16248.272,E2 16248.272} C_VEL
LIN {X 0,Y 449.122,Z 256.785,A -85,B 0,C 180,E1 16244.527,E2 16244.527} C_VEL
LIN {X 0,Y 449.114,Z 256.774,A -85,B 0,C 180,E1 16240.808,E2 16240.808} C_VEL
LIN {X 0,Y 449.122,Z 256.778,A -85,B 0,C 180,E1 16237.106,E2 16237.106} C_VEL
LIN {X 0,Y 449.134,Z 256.79,A -85,B 0,C 180,E1 16233.356,E2 16233.356} C_VEL
LIN {X 0,Y 449.132,Z 256.775,A -85,B 0,C 180,E1 16229.616,E2 16229.616} C_VEL
LIN {X 0,Y 449.132,Z 256.775,A -85,B 0,C 180,E1 16225.869,E2 16225.869} C_VEL
LIN {X 0,Y 449.124,Z 256.787,A -85,B 0,C 180,E1 16222.099,E2 16222.099} C_VEL
LIN {X 0,Y 449.112,Z 256.782,A -85,B 0,C 180,E1 16218.428,E2 16218.428} C_VEL
LIN {X 0,Y 449.116,Z 256.771,A -85,B 0,C 180,E1 16214.701,E2 16214.701} C_VEL
LIN {X 0,Y 449.131,Z 256.791,A -85,B 0,C 180,E1 16210.971,E2 16210.971} C_VEL
LIN {X 0,Y 449.136,Z 256.774,A -85,B 0,C 180,E1 16207.289,E2 16207.289} C_VEL
LIN {X 0,Y 449.129,Z 256.776,A -85,B 0,C 180,E1 16203.573,E2 16203.573} C_VEL
LIN {X 0,Y 449.114,Z 256.788,A -85,B 0,C 180,E1 16199.871,E2 16199.871} C_VEL
LIN {X 0,Y 449.11,Z 256.786,A -85,B 0,C 180,E1 16196.169,E2 16196.169} C_VEL
LIN {X 0,Y 449.119,Z 256.773,A -85,B 0,C 180,E1 16192.451,E2 16192.451} C_VEL
LIN {X 0,Y 449.132,Z 256.778,A -85,B 0,C 180,E1 16188.701,E2 16188.701} C_VEL
LIN {X 0,Y 449.14,Z 256.79,A -85,B 0,C 180,E1 16184.902,E2 16184.902} C_VEL
LIN {X 0,Y 449.134,Z 256.788,A -85,B 0,C 180,E1 16181.102,E2 16181.102} C_VEL
LIN {X 0,Y 449.119,Z 256.788,A -85,B 0,C 180,E1 16177.347,E2 16177.347} C_VEL
LIN {X 0,Y 449.108,Z 256.791,A -85,B 0,C 180,E1 16173.701,E2 16173.701} C_VEL
LIN {X 0,Y 449.112,Z 256.793,A -85,B 0,C 180,E1 16169.939,E2 16169.939} C_VEL
LIN {X 0,Y 449.131,Z 256.793,A -85,B 0,C 180,E1 16166.335,E2 16166.335} C_VEL
LIN {X 0,Y 449.139,Z 256.781,A -85,B 0,C 180,E1 16162.573,E2 16162.573} C_VEL
LIN {X 0,Y 449.152,Z 257.06,A -85,B 0,C 180,E1 16159.867,E2 16159.867} C_VEL
LIN {X 0,Y 450.572,Z 260.493,A -85,B 0,C 180,E1 16159.276,E2 16159.276} C_VEL
LIN {X 0,Y 451.749,Z 262.749,A -85,B 0,C 180,E1 16158.901,E2 16158.901} C_VEL
LIN {X 0,Y 459.282,Z 277.888,A -85,B 0,C 180,E1 16156.533,E2 16156.533} C_VEL
LIN {X 0,Y 468.568,Z 298.413,A -85,B 0,C 180,E1 16153.665,E2 16153.665} C_VEL
LIN {X 0,Y 470.751,Z 303.076,A -85,B 0,C 180,E1 16153.126,E2 16153.126} C_VEL
LIN {X 0,Y 474.363,Z 309.631,A -85,B 0,C 180,E1 16152.629,E2 16152.629} C_VEL
LIN {X 0,Y 477.422,Z 331.713,A -85,B 0,C 180,E1 16151.901,E2 16151.901} C_VEL
LIN {X 0,Y 472.767,Z 547.328,A -85,B 0,C 180,E1 16148.298,E2 16148.298} C_VEL
LIN {X 0,Y 471.4,Z 607.414,A -85,B 0,C 180,E1 16147.277,E2 16147.277} C_VEL
LIN {X 0,Y 470.186,Z 629.029,A -85,B 0,C 180,E1 16146.705,E2 16146.705} C_VEL
LIN {X 0,Y 468.574,Z 651.097,A -85,B 0,C 180,E1 16145.894,E2 16145.894} C_VEL
LIN {X 0,Y 466.804,Z 671.155,A -85,B 0,C 180,E1 16144.949,E2 16144.949} C_VEL
LIN {X 0,Y 464.803,Z 690.87,A -85,B 0,C 180,E1 16143.782,E2 16143.782} C_VEL
LIN {X 0,Y 462.502,Z 711.111,A -85,B 0,C 180,E1 16142.338,E2 16142.338} C_VEL
LIN {X 0,Y 460.314,Z 729.525,A -85,B 0,C 180,E1 16140.778,E2 16140.778} C_VEL
LIN {X 0,Y 458.066,Z 747.454,A -85,B 0,C 180,E1 16138.983,E2 16138.983} C_VEL
LIN {X 0,Y 455.932,Z 764.396,A -85,B 0,C 180,E1 16136.996,E2 16136.996} C_VEL
LIN {X 0,Y 453.991,Z 780.134,A -85,B 0,C 180,E1 16134.854,E2 16134.854} C_VEL
LIN {X 0,Y 452.338,Z 794.247,A -85,B 0,C 180,E1 16132.618,E2 16132.618} C_VEL
LIN {X 0,Y 450.942,Z 807.098,A -85,B 0,C 180,E1 16130.235,E2 16130.235} C_VEL
LIN {X 0,Y 449.912,Z 817.281,A -85,B 0,C 180,E1 16127.98,E2 16127.98} C_VEL
LIN {X 0,Y 449.034,Z 827.055,A -85,B 0,C 180,E1 16125.364,E2 16125.364} C_VEL
LIN {X 0,Y 448.446,Z 835.471,A -85,B 0,C 180,E1 16122.619,E2 16122.619} C_VEL
LIN {X 0,Y 448.121,Z 842.132,A -85,B 0,C 180,E1 16119.891,E2 16119.891} C_VEL
LIN {X 0,Y 447.98,Z 846.814,A -85,B 0,C 180,E1 16117.308,E2 16117.308} C_VEL
LIN {X 0,Y 447.921,Z 850.332,A -85,B 0,C 180,E1 16114.48,E2 16114.48} C_VEL
LIN {X 0,Y 447.904,Z 852.086,A -85,B 0,C 180,E1 16111.918,E2 16111.918} C_VEL
LIN {X 0,Y 447.902,Z 852.371,A -85,B 0,C 180,E1 16109.231,E2 16109.231} C_VEL
LIN {X 0,Y 447.912,Z 851.234,A -85,B 0,C 180,E1 16106.543,E2 16106.543} C_VEL
LIN {X 0,Y 447.941,Z 848.614,A -85,B 0,C 180,E1 16103.977,E2 16103.977} C_VEL
LIN {X 0,Y 448.034,Z 844.412,A -85,B 0,C 180,E1 16101.27,E2 16101.27} C_VEL
LIN {X 0,Y 448.263,Z 838.853,A -85,B 0,C 180,E1 16098.679,E2 16098.679} C_VEL
LIN {X 0,Y 448.717,Z 831.28,A -85,B 0,C 180,E1 16095.942,E2 16095.942} C_VEL
LIN {X 0,Y 449.436,Z 822.371,A -85,B 0,C 180,E1 16093.321,E2 16093.321} C_VEL
LIN {X 0,Y 450.435,Z 812.083,A -85,B 0,C 180,E1 16090.82,E2 16090.82} C_VEL
LIN {X 0,Y 451.588,Z 800.878,A -85,B 0,C 180,E1 16088.571,E2 16088.571} C_VEL
LIN {X 0,Y 453.172,Z 786.903,A -85,B 0,C 180,E1 16086.185,E2 16086.185} C_VEL
LIN {X 0,Y 455.027,Z 771.309,A -85,B 0,C 180,E1 16083.929,E2 16083.929} C_VEL
LIN {X 0,Y 456.998,Z 755.339,A -85,B 0,C 180,E1 16081.939,E2 16081.939} C_VEL
LIN {X 0,Y 459.129,Z 738.109,A -85,B 0,C 180,E1 16080.082,E2 16080.082} C_VEL
LIN {X 0,Y 461.411,Z 719.331,A -85,B 0,C 180,E1 16078.371,E2 16078.371} C_VEL
LIN {X 0,Y 463.626,Z 699.658,A -85,B 0,C 180,E1 16076.858,E2 16076.858} C_VEL
LIN {X 0,Y 465.803,Z 679.242,A -85,B 0,C 180,E1 16075.554,E2 16075.554} C_VEL
LIN {X 0,Y 467.655,Z 659.443,A -85,B 0,C 180,E1 16074.523,E2 16074.523} C_VEL
LIN {X 0,Y 469.303,Z 637.976,A -85,B 0,C 180,E1 16073.643,E2 16073.643} C_VEL
LIN {X 0,Y 470.742,Z 615.335,A -85,B 0,C 180,E1 16072.961,E2 16072.961} C_VEL
LIN {X 0,Y 471.607,Z 592.987,A -85,B 0,C 180,E1 16072.501,E2 16072.501} C_VEL
LIN {X 0,Y 476.223,Z 366.783,A -85,B 0,C 180,E1 16068.755,E2 16068.755} C_VEL
LIN {X 0,Y 476.872,Z 329.393,A -85,B 0,C 180,E1 16068.102,E2 16068.102} C_VEL
LIN {X 0,Y 473.696,Z 308.438,A -85,B 0,C 180,E1 16067.381,E2 16067.381} C_VEL
LIN {X 0,Y 469.693,Z 301.426,A -85,B 0,C 180,E1 16066.811,E2 16066.811} C_VEL
LIN {X 0,Y 461.878,Z 283.469,A -85,B 0,C 180,E1 16064.365,E2 16064.365} C_VEL
LIN {X 0,Y 455.252,Z 269.508,A -85,B 0,C 180,E1 16062.227,E2 16062.227} C_VEL
LIN {X 0,Y 451.125,Z 261.168,A -85,B 0,C 180,E1 16060.831,E2 16060.831} C_VEL
LIN {X 0,Y 449.377,Z 258.017,A -85,B 0,C 180,E1 16060.254,E2 16060.254} C_VEL
LIN {X 0,Y 449.14,Z 256.825,A -85,B 0,C 180,E1 16059.938,E2 16059.938} C_VEL
LIN {X 0,Y 449.126,Z 256.786,A -85,B 0,C 180,E1 16056.154,E2 16056.154} C_VEL
LIN {X 0,Y 449.123,Z 256.791,A -85,B 0,C 180,E1 16052.448,E2 16052.448} C_VEL
LIN {X 0,Y 449.129,Z 256.782,A -85,B 0,C 180,E1 16048.7,E2 16048.7} C_VEL
LIN {X 0,Y 449.134,Z 256.789,A -85,B 0,C 180,E1 16045.023,E2 16045.023} C_VEL
LIN {X 0,Y 449.124,Z 256.785,A -85,B 0,C 180,E1 16041.278,E2 16041.278} C_VEL
LIN {X 0,Y 449.119,Z 256.782,A -85,B 0,C 180,E1 16037.491,E2 16037.491} C_VEL
LIN {X 0,Y 449.128,Z 256.783,A -85,B 0,C 180,E1 16033.782,E2 16033.782} C_VEL
LIN {X 0,Y 449.132,Z 256.785,A -85,B 0,C 180,E1 16030.001,E2 16030.001} C_VEL
LIN {X 0,Y 449.138,Z 256.789,A -85,B 0,C 180,E1 16026.263,E2 16026.263} C_VEL
LIN {X 0,Y 449.131,Z 256.79,A -85,B 0,C 180,E1 16022.553,E2 16022.553} C_VEL
LIN {X 0,Y 449.103,Z 256.788,A -85,B 0,C 180,E1 16018.981,E2 16018.981} C_VEL
LIN {X 0,Y 449.098,Z 256.787,A -85,B 0,C 180,E1 16015.276,E2 16015.276} C_VEL
LIN {X 0,Y 449.114,Z 256.794,A -85,B 0,C 180,E1 16011.681,E2 16011.681} C_VEL
LIN {X 0,Y 449.129,Z 256.785,A -85,B 0,C 180,E1 16007.922,E2 16007.922} C_VEL
LIN {X 0,Y 449.132,Z 256.791,A -85,B 0,C 180,E1 16004.242,E2 16004.242} C_VEL
LIN {X 0,Y 449.12,Z 257.052,A -85,B 0,C 180,E1 16001.192,E2 16001.192} C_VEL
LIN {X 0,Y 450.415,Z 260.297,A -85,B 0,C 180,E1 16000.552,E2 16000.552} C_VEL
LIN {X 0,Y 451.402,Z 262.109,A -85,B 0,C 180,E1 16000.192,E2 16000.192} C_VEL
LIN {X 0,Y 456.946,Z 274.185,A -85,B 0,C 180,E1 15998.028,E2 15998.028} C_VEL
LIN {X 0,Y 463.215,Z 288.683,A -85,B 0,C 180,E1 15995.654,E2 15995.654} C_VEL
LIN {X 0,Y 467.841,Z 300.281,A -85,B 0,C 180,E1 15993.949,E2 15993.949} C_VEL
LIN {X 0,Y 470.107,Z 304.739,A -85,B 0,C 180,E1 15993.609,E2 15993.609} C_VEL
LIN {X 0,Y 474.168,Z 328.579,A -85,B 0,C 180,E1 15992.692,E2 15992.692} C_VEL
LIN {X 0,Y 467.989,Z 565.974,A -85,B 0,C 180,E1 15988.58,E2 15988.58} C_VEL
LIN {X 0,Y 466.911,Z 586.886,A -85,B 0,C 180,E1 15987.99,E2 15987.99} C_VEL
LIN {X 0,Y 465.602,Z 605.878,A -85,B 0,C 180,E1 15987.239,E2 15987.239} C_VEL
LIN {X 0,Y 463.887,Z 625.859,A -85,B 0,C 180,E1 15986.216,E2 15986.216} C_VEL
LIN {X 0,Y 461.998,Z 644.635,A -85,B 0,C 180,E1 15985.006,E2 15985.006} C_VEL
LIN {X 0,Y 460.089,Z 661.81,A -85,B 0,C 180,E1 15983.661,E2 15983.661} C_VEL
LIN {X 0,Y 459.254,Z 668.616,A -85,B 0,C 180,E1 15983.048,E2 15983.048} C_VEL
LIN {X 0,Y 457.624,Z 674.913,A -85,B 0,C 180,E1 15982.516,E2 15982.516} C_VEL
LIN {X 0,Y 450.215,Z 690.637,A -85,B 0,C 180,E1 15981.217,E2 15981.217} C_VEL
LIN {X 0,Y 448.56,Z 696.282,A -85,B 0,C 180,E1 15980.59,E2 15980.59} C_VEL
LIN {X 0,Y 446.555,Z 710.749,A -85,B 0,C 180,E1 15978.599,E2 15978.599} C_VEL
LIN {X 0,Y 444.714,Z 724.297,A -85,B 0,C 180,E1 15976.384,E2 15976.384} C_VEL
LIN {X 0,Y 443.144,Z 736.61,A -85,B 0,C 180,E1 15973.968,E2 15973.968} C_VEL
LIN {X 0,Y 441.953,Z 746.962,A -85,B 0,C 180,E1 15971.512,E2 15971.512} C_VEL
LIN {X 0,Y 441.103,Z 755.709,A -85,B 0,C 180,E1 15968.972,E2 15968.972} C_VEL
LIN {X 0,Y 440.539,Z 762.931,A -85,B 0,C 180,E1 15966.324,E2 15966.324} C_VEL
LIN {X 0,Y 440.222,Z 768.361,A -85,B 0,C 180,E1 15963.656,E2 15963.656} C_VEL
LIN {X 0,Y 440.076,Z 772.05,A -85,B 0,C 180,E1 15961.049,E2 15961.049} C_VEL
LIN {X 0,Y 440.028,Z 774.27,A -85,B 0,C 180,E1 15958.354,E2 15958.354} C_VEL
LIN {X 0,Y 440.011,Z 774.906,A -85,B 0,C 180,E1 15955.724,E2 15955.724} C_VEL
LIN {X 0,Y 440.029,Z 773.966,A -85,B 0,C 180,E1 15953.04,E2 15953.04} C_VEL
LIN {X 0,Y 440.086,Z 771.351,A -85,B 0,C 180,E1 15950.342,E2 15950.342} C_VEL
LIN {X 0,Y 440.247,Z 767.223,A -85,B 0,C 180,E1 15947.719,E2 15947.719} C_VEL
LIN {X 0,Y 440.603,Z 761.201,A -85,B 0,C 180,E1 15944.994,E2 15944.994} C_VEL
LIN {X 0,Y 441.207,Z 753.684,A -85,B 0,C 180,E1 15942.395,E2 15942.395} C_VEL
LIN {X 0,Y 442.103,Z 744.674,A -85,B 0,C 180,E1 15939.898,E2 15939.898} C_VEL
LIN {X 0,Y 443.383,Z 733.556,A -85,B 0,C 180,E1 15937.386,E2 15937.386} C_VEL
LIN {X 0,Y 444.979,Z 720.898,A -85,B 0,C 180,E1 15935.029,E2 15935.029} C_VEL
LIN {X 0,Y 446.745,Z 707.586,A -85,B 0,C 180,E1 15932.952,E2 15932.952} C_VEL
LIN {X 0,Y 448.784,Z 692.459,A -85,B 0,C 180,E1 15930.959,E2 15930.959} C_VEL
LIN {X 0,Y 450.987,Z 675.73,A -85,B 0,C 180,E1 15929.112,E2 15929.112} C_VEL
LIN {X 0,Y 453.137,Z 658.612,A -85,B 0,C 180,E1 15927.535,E2 15927.535} C_VEL
LIN {X 0,Y 455.217,Z 640.632,A -85,B 0,C 180,E1 15926.16,E2 15926.16} C_VEL
LIN {X 0,Y 457.152,Z 621.622,A -85,B 0,C 180,E1 15924.982,E2 15924.982} C_VEL
LIN {X 0,Y 458.767,Z 602.133,A -85,B 0,C 180,E1 15924.028,E2 15924.028} C_VEL
LIN {X 0,Y 460.143,Z 581.943,A -85,B 0,C 180,E1 15923.282,E2 15923.282} C_VEL
LIN {X 0,Y 461.128,Z 560.619,A -85,B 0,C 180,E1 15922.734,E2 15922.734} C_VEL
LIN {X 0,Y 466.961,Z 328.666,A -85,B 0,C 180,E1 15918.741,E2 15918.741} C_VEL
LIN {X 0,Y 462.765,Z 306.259,A -85,B 0,C 180,E1 15917.863,E2 15917.863} C_VEL
LIN {X 0,Y 458.857,Z 299.392,A -85,B 0,C 180,E1 15917.288,E2 15917.288} C_VEL
LIN {X 0,Y 451.395,Z 280.81,A -85,B 0,C 180,E1 15914.455,E2 15914.455} C_VEL
LIN {X 0,Y 444.227,Z 264.971,A -85,B 0,C 180,E1 15911.768,E2 15911.768} C_VEL
LIN {X 0,Y 441.228,Z 257.998,A -85,B 0,C 180,E1 15910.502,E2 15910.502} C_VEL
LIN {X 0,Y 441.185,Z 257.727,A -85,B 0,C 180,E1 15906.777,E2 15906.777} C_VEL
LIN {X 0,Y 441.182,Z 257.78,A -85,B 0,C 180,E1 15902.952,E2 15902.952} C_VEL
LIN {X 0,Y 441.18,Z 257.776,A -85,B 0,C 180,E1 15899.192,E2 15899.192} C_VEL
LIN {X 0,Y 441.189,Z 257.773,A -85,B 0,C 180,E1 15895.491,E2 15895.491} C_VEL
LIN {X 0,Y 441.199,Z 257.774,A -85,B 0,C 180,E1 15891.617,E2 15891.617} C_VEL
LIN {X 0,Y 441.194,Z 257.78,A -85,B 0,C 180,E1 15887.82,E2 15887.82} C_VEL
LIN {X 0,Y 441.197,Z 257.773,A -85,B 0,C 180,E1 15884.08,E2 15884.08} C_VEL
LIN {X 0,Y 441.194,Z 257.764,A -85,B 0,C 180,E1 15880.23,E2 15880.23} C_VEL
LIN {X 0,Y 441.176,Z 257.763,A -85,B 0,C 180,E1 15876.586,E2 15876.586} C_VEL
LIN {X 0,Y 441.177,Z 257.776,A -85,B 0,C 180,E1 15872.777,E2 15872.777} C_VEL
LIN {X 0,Y 441.187,Z 257.774,A -85,B 0,C 180,E1 15868.984,E2 15868.984} C_VEL
LIN {X 0,Y 441.192,Z 257.759,A -85,B 0,C 180,E1 15865.216,E2 15865.216} C_VEL
LIN {X 0,Y 441.198,Z 257.774,A -85,B 0,C 180,E1 15861.398,E2 15861.398} C_VEL
LIN {X 0,Y 441.197,Z 257.772,A -85,B 0,C 180,E1 15857.541,E2 15857.541} C_VEL
LIN {X 0,Y 441.192,Z 257.753,A -85,B 0,C 180,E1 15853.765,E2 15853.765} C_VEL
LIN {X 0,Y 441.177,Z 257.773,A -85,B 0,C 180,E1 15850.049,E2 15850.049} C_VEL
LIN {X 0,Y 441.172,Z 257.78,A -85,B 0,C 180,E1 15846.244,E2 15846.244} C_VEL
LIN {X 0,Y 441.174,Z 257.762,A -85,B 0,C 180,E1 15842.467,E2 15842.467} C_VEL
LIN {X 0,Y 441.194,Z 257.767,A -85,B 0,C 180,E1 15838.83,E2 15838.83} C_VEL
LIN {X 0,Y 441.197,Z 257.776,A -85,B 0,C 180,E1 15835.059,E2 15835.059} C_VEL
LIN {X 0,Y 441.197,Z 257.766,A -85,B 0,C 180,E1 15831.266,E2 15831.266} C_VEL
LIN {X 0,Y 441.177,Z 257.759,A -85,B 0,C 180,E1 15827.566,E2 15827.566} C_VEL
LIN {X 0,Y 441.169,Z 257.77,A -85,B 0,C 180,E1 15823.928,E2 15823.928} C_VEL
LIN {X 0,Y 441.174,Z 257.775,A -85,B 0,C 180,E1 15820.125,E2 15820.125} C_VEL
LIN {X 0,Y 441.196,Z 257.778,A -85,B 0,C 180,E1 15816.492,E2 15816.492} C_VEL
LIN {X 0,Y 441.202,Z 257.777,A -85,B 0,C 180,E1 15812.663,E2 15812.663} C_VEL
LIN {X 0,Y 441.201,Z 257.773,A -85,B 0,C 180,E1 15808.888,E2 15808.888} C_VEL
LIN {X 0,Y 441.184,Z 257.769,A -85,B 0,C 180,E1 15805.122,E2 15805.122} C_VEL
LIN {X 0,Y 441.166,Z 257.774,A -85,B 0,C 180,E1 15801.432,E2 15801.432} C_VEL
LIN {X 0,Y 441.248,Z 258.117,A -85,B 0,C 180,E1 15800.835,E2 15800.835} C_VEL
LIN {X 0,Y 442.632,Z 261.442,A -85,B 0,C 180,E1 15800.262,E2 15800.262} C_VEL
LIN {X 0,Y 443.775,Z 263.654,A -85,B 0,C 180,E1 15799.88,E2 15799.88} C_VEL
LIN {X 0,Y 448.019,Z 272.04,A -85,B 0,C 180,E1 15798.484,E2 15798.484} C_VEL
LIN {X 0,Y 455.939,Z 288.476,A -85,B 0,C 180,E1 15795.959,E2 15795.959} C_VEL
LIN {X 0,Y 462.146,Z 302.286,A -85,B 0,C 180,E1 15794.064,E2 15794.064} C_VEL
LIN {X 0,Y 468.547,Z 313.419,A -85,B 0,C 180,E1 15793.151,E2 15793.151} C_VEL
LIN {X 0,Y 471.196,Z 333.196,A -85,B 0,C 180,E1 15792.492,E2 15792.492} C_VEL
LIN {X 0,Y 466.25,Z 548.58,A -85,B 0,C 180,E1 15788.852,E2 15788.852} C_VEL
LIN {X 0,Y 464.831,Z 607.202,A -85,B 0,C 180,E1 15787.843,E2 15787.843} C_VEL
LIN {X 0,Y 463.542,Z 628.984,A -85,B 0,C 180,E1 15787.259,E2 15787.259} C_VEL
LIN {X 0,Y 461.872,Z 650.579,A -85,B 0,C 180,E1 15786.456,E2 15786.456} C_VEL
LIN {X 0,Y 459.95,Z 671.073,A -85,B 0,C 180,E1 15785.478,E2 15785.478} C_VEL
LIN {X 0,Y 457.82,Z 690.823,A -85,B 0,C 180,E1 15784.293,E2 15784.293} C_VEL
LIN {X 0,Y 455.402,Z 710.885,A -85,B 0,C 180,E1 15782.838,E2 15782.838} C_VEL
LIN {X 0,Y 452.993,Z 729.819,A -85,B 0,C 180,E1 15781.202,E2 15781.202} C_VEL
LIN {X 0,Y 450.609,Z 747.824,A -85,B 0,C 180,E1 15779.364,E2 15779.364} C_VEL
LIN {X 0,Y 448.345,Z 764.605,A -85,B 0,C 180,E1 15777.347,E2 15777.347} C_VEL
LIN {X 0,Y 446.192,Z 780.955,A -85,B 0,C 180,E1 15775.055,E2 15775.055} C_VEL
LIN {X 0,Y 444.426,Z 795.266,A -85,B 0,C 180,E1 15772.719,E2 15772.719} C_VEL
LIN {X 0,Y 442.933,Z 808.314,A -85,B 0,C 180,E1 15770.203,E2 15770.203} C_VEL
LIN {X 0,Y 441.799,Z 819.539,A -85,B 0,C 180,E1 15767.652,E2 15767.652} C_VEL
LIN {X 0,Y 441.071,Z 827.972,A -85,B 0,C 180,E1 15765.379,E2 15765.379} C_VEL
LIN {X 0,Y 440.479,Z 835.824,A -85,B 0,C 180,E1 15762.718,E2 15762.718} C_VEL
LIN {X 0,Y 440.131,Z 842.386,A -85,B 0,C 180,E1 15759.941,E2 15759.941} C_VEL
LIN {X 0,Y 439.983,Z 847.021,A -85,B 0,C 180,E1 15757.31,E2 15757.31} C_VEL
LIN {X 0,Y 439.92,Z 850.445,A -85,B 0,C 180,E1 15754.431,E2 15754.431} C_VEL
LIN {X 0,Y 439.899,Z 852.209,A -85,B 0,C 180,E1 15751.692,E2 15751.692} C_VEL
LIN {X 0,Y 439.906,Z 852.347,A -85,B 0,C 180,E1 15749.087,E2 15749.087} C_VEL
LIN {X 0,Y 439.91,Z 851.122,A -85,B 0,C 180,E1 15746.35,E2 15746.35} C_VEL
LIN {X 0,Y 439.945,Z 848.454,A -85,B 0,C 180,E1 15743.736,E2 15743.736} C_VEL
LIN {X 0,Y 440.071,Z 843.904,A -85,B 0,C 180,E1 15740.847,E2 15740.847} C_VEL
LIN {X 0,Y 440.361,Z 837.932,A -85,B 0,C 180,E1 15738.074,E2 15738.074} C_VEL
LIN {X 0,Y 440.856,Z 830.469,A -85,B 0,C 180,E1 15735.418,E2 15735.418} C_VEL
LIN {X 0,Y 441.562,Z 822.212,A -85,B 0,C 180,E1 15733.015,E2 15733.015} C_VEL
LIN {X 0,Y 442.608,Z 811.4,A -85,B 0,C 180,E1 15730.467,E2 15730.467} C_VEL
LIN {X 0,Y 443.917,Z 799.275,A -85,B 0,C 180,E1 15728.043,E2 15728.043} C_VEL
LIN {X 0,Y 445.63,Z 785.113,A -85,B 0,C 180,E1 15725.615,E2 15725.615} C_VEL
LIN {X 0,Y 447.57,Z 769.888,A -85,B 0,C 180,E1 15723.389,E2 15723.389} C_VEL
LIN {X 0,Y 449.758,Z 753.193,A -85,B 0,C 180,E1 15721.301,E2 15721.301} C_VEL
LIN {X 0,Y 452.184,Z 734.785,A -85,B 0,C 180,E1 15719.334,E2 15719.334} C_VEL
LIN {X 0,Y 454.595,Z 716.024,A -85,B 0,C 180,E1 15717.628,E2 15717.628} C_VEL
LIN {X 0,Y 456.898,Z 696.695,A -85,B 0,C 180,E1 15716.163,E2 15716.163} C_VEL
LIN {X 0,Y 459.095,Z 676.713,A -85,B 0,C 180,E1 15714.902,E2 15714.902} C_VEL
LIN {X 0,Y 461.086,Z 656.452,A -85,B 0,C 180,E1 15713.854,E2 15713.854} C_VEL
LIN {X 0,Y 462.822,Z 634.989,A -85,B 0,C 180,E1 15712.997,E2 15712.997} C_VEL
LIN {X 0,Y 464.22,Z 613.082,A -85,B 0,C 180,E1 15712.355,E2 15712.355} C_VEL
LIN {X 0,Y 465.093,Z 589.393,A -85,B 0,C 180,E1 15711.882,E2 15711.882} C_VEL
LIN {X 0,Y 470.008,Z 365.3,A -85,B 0,C 180,E1 15708.122,E2 15708.122} C_VEL
LIN {X 0,Y 470.651,Z 330.872,A -85,B 0,C 180,E1 15707.513,E2 15707.513} C_VEL
LIN {X 0,Y 467.818,Z 312.17,A -85,B 0,C 180,E1 15706.852,E2 15706.852} C_VEL
LIN {X 0,Y 461.642,Z 301.546,A -85,B 0,C 180,E1 15705.952,E2 15705.952} C_VEL
LIN {X 0,Y 453.47,Z 282.949,A -85,B 0,C 180,E1 15703.293,E2 15703.293} C_VEL
LIN {X 0,Y 446.948,Z 269.781,A -85,B 0,C 180,E1 15701.125,E2 15701.125} C_VEL
LIN {X 0,Y 445.107,Z 266.111,A -85,B 0,C 180,E1 15700.481,E2 15700.481} C_VEL
LIN {X 0,Y 442.928,Z 261.835,A -85,B 0,C 180,E1 15699.706,E2 15699.706} C_VEL
LIN {X 0,Y 441.252,Z 258.159,A -85,B 0,C 180,E1 15699.004,E2 15699.004} C_VEL
LIN {X 0,Y 441.181,Z 257.776,A -85,B 0,C 180,E1 15698.357,E2 15698.357} C_VEL
LIN {X 0,Y 441.184,Z 257.777,A -85,B 0,C 180,E1 15694.513,E2 15694.513} C_VEL
LIN {X 0,Y 441.192,Z 257.777,A -85,B 0,C 180,E1 15690.804,E2 15690.804} C_VEL
LIN {X 0,Y 441.197,Z 257.775,A -85,B 0,C 180,E1 15687.045,E2 15687.045} C_VEL
LIN {X 0,Y 441.187,Z 257.772,A -85,B 0,C 180,E1 15683.225,E2 15683.225} C_VEL
LIN {X 0,Y 441.183,Z 257.78,A -85,B 0,C 180,E1 15679.461,E2 15679.461} C_VEL
LIN {X 0,Y 441.183,Z 257.78,A -85,B 0,C 180,E1 15675.647,E2 15675.647} C_VEL
LIN {X 0,Y 441.191,Z 257.773,A -85,B 0,C 180,E1 15671.902,E2 15671.902} C_VEL
LIN {X 0,Y 441.2,Z 257.77,A -85,B 0,C 180,E1 15668.078,E2 15668.078} C_VEL
LIN {X 0,Y 441.197,Z 257.769,A -85,B 0,C 180,E1 15664.29,E2 15664.29} C_VEL
LIN {X 0,Y 441.195,Z 257.774,A -85,B 0,C 180,E1 15660.52,E2 15660.52} C_VEL
LIN {X 0,Y 441.174,Z 257.781,A -85,B 0,C 180,E1 15656.753,E2 15656.753} C_VEL
LIN {X 0,Y 441.155,Z 257.775,A -85,B 0,C 180,E1 15653.083,E2 15653.083} C_VEL
LIN {X 0,Y 441.155,Z 257.784,A -85,B 0,C 180,E1 15649.291,E2 15649.291} C_VEL
LIN {X 0,Y 441.163,Z 257.777,A -85,B 0,C 180,E1 15645.565,E2 15645.565} C_VEL
LIN {X 0,Y 441.217,Z 258.034,A -85,B 0,C 180,E1 15642.291,E2 15642.291} C_VEL
LIN {X 0,Y 442.738,Z 261.642,A -85,B 0,C 180,E1 15641.536,E2 15641.536} C_VEL
LIN {X 0,Y 447.26,Z 270.927,A -85,B 0,C 180,E1 15639.728,E2 15639.728} C_VEL
LIN {X 0,Y 453.997,Z 286.131,A -85,B 0,C 180,E1 15637.059,E2 15637.059} C_VEL
LIN {X 0,Y 459.828,Z 300.408,A -85,B 0,C 180,E1 15634.845,E2 15634.845} C_VEL
LIN {X 0,Y 464.485,Z 308.703,A -85,B 0,C 180,E1 15634.139,E2 15634.139} C_VEL
LIN {X 0,Y 468.032,Z 330.073,A -85,B 0,C 180,E1 15633.301,E2 15633.301} C_VEL
LIN {X 0,Y 461.451,Z 566.379,A -85,B 0,C 180,E1 15629.146,E2 15629.146} C_VEL
LIN {X 0,Y 460.323,Z 587.21,A -85,B 0,C 180,E1 15628.552,E2 15628.552} C_VEL
LIN {X 0,Y 458.92,Z 606.533,A -85,B 0,C 180,E1 15627.781,E2 15627.781} C_VEL
LIN {X 0,Y 457.09,Z 626.725,A -85,B 0,C 180,E1 15626.731,E2 15626.731} C_VEL
LIN {X 0,Y 455.056,Z 645.75,A -85,B 0,C 180,E1 15625.484,E2 15625.484} C_VEL
LIN {X 0,Y 453.001,Z 663.053,A -85,B 0,C 180,E1 15624.101,E2 15624.101} C_VEL
LIN {X 0,Y 450.728,Z 680.577,A -85,B 0,C 180,E1 15622.41,E2 15622.41} C_VEL
LIN {X 0,Y 448.56,Z 696.282,A -85,B 0,C 180,E1 15620.59,E2 15620.59} C_VEL
LIN {X 0,Y 446.913,Z 701.876,A -85,B 0,C 180,E1 15619.934,E2 15619.934} C_VEL
LIN {X 0,Y 439.457,Z 715.704,A -85,B 0,C 180,E1 15618.297,E2 15618.297} C_VEL
LIN {X 0,Y 437.834,Z 720.618,A -85,B 0,C 180,E1 15617.55,E2 15617.55} C_VEL
LIN {X 0,Y 436.1,Z 732.836,A -85,B 0,C 180,E1 15615.264,E2 15615.264} C_VEL
LIN {X 0,Y 434.665,Z 743.83,A -85,B 0,C 180,E1 15612.797,E2 15612.797} C_VEL
LIN {X 0,Y 433.583,Z 753.26,A -85,B 0,C 180,E1 15610.219,E2 15610.219} C_VEL
LIN {X 0,Y 432.849,Z 761.018,A -85,B 0,C 180,E1 15607.578,E2 15607.578} C_VEL
LIN {X 0,Y 432.419,Z 766.948,A -85,B 0,C 180,E1 15604.991,E2 15604.991} C_VEL
LIN {X 0,Y 432.179,Z 771.373,A -85,B 0,C 180,E1 15602.306,E2 15602.306} C_VEL
LIN {X 0,Y 432.083,Z 774.155,A -85,B 0,C 180,E1 15599.685,E2 15599.685} C_VEL
LIN {X 0,Y 432.047,Z 775.509,A -85,B 0,C 180,E1 15596.975,E2 15596.975} C_VEL
LIN {X 0,Y 432.053,Z 775.309,A -85,B 0,C 180,E1 15594.25,E2 15594.25} C_VEL
LIN {X 0,Y 432.082,Z 773.503,A -85,B 0,C 180,E1 15591.532,E2 15591.532} C_VEL
LIN {X 0,Y 432.206,Z 770.168,A -85,B 0,C 180,E1 15588.89,E2 15588.89} C_VEL
LIN {X 0,Y 432.489,Z 764.983,A -85,B 0,C 180,E1 15586.108,E2 15586.108} C_VEL
LIN {X 0,Y 433.035,Z 758.023,A -85,B 0,C 180,E1 15583.351,E2 15583.351} C_VEL
LIN {X 0,Y 433.858,Z 749.685,A -85,B 0,C 180,E1 15580.76,E2 15580.76} C_VEL
LIN {X 0,Y 434.99,Z 740.097,A -85,B 0,C 180,E1 15578.328,E2 15578.328} C_VEL
LIN {X 0,Y 436.487,Z 728.554,A -85,B 0,C 180,E1 15575.918,E2 15575.918} C_VEL
LIN {X 0,Y 438.284,Z 715.623,A -85,B 0,C 180,E1 15573.664,E2 15573.664} C_VEL
LIN {X 0,Y 440.336,Z 701.297,A -85,B 0,C 180,E1 15571.563,E2 15571.563} C_VEL
LIN {X 0,Y 442.595,Z 685.472,A -85,B 0,C 180,E1 15569.613,E2 15569.613} C_VEL
LIN {X 0,Y 444.816,Z 669.327,A -85,B 0,C 180,E1 15567.94,E2 15567.94} C_VEL
LIN {X 0,Y 447.097,Z 651.657,A -85,B 0,C 180,E1 15566.411,E2 15566.411} C_VEL
LIN {X 0,Y 449.253,Z 632.892,A -85,B 0,C 180,E1 15565.086,E2 15565.086} C_VEL
LIN {X 0,Y 451.1,Z 614.162,A -85,B 0,C 180,E1 15564.022,E2 15564.022} C_VEL
LIN {X 0,Y 452.759,Z 593.75,A -85,B 0,C 180,E1 15563.117,E2 15563.117} C_VEL
LIN {X 0,Y 454.052,Z 572.698,A -85,B 0,C 180,E1 15562.437,E2 15562.437} C_VEL
LIN {X 0,Y 454.909,Z 550.33,A -85,B 0,C 180,E1 15561.963,E2 15561.963} C_VEL
LIN {X 0,Y 460.733,Z 330.138,A -85,B 0,C 180,E1 15558.135,E2 15558.135} C_VEL
LIN {X 0,Y 457.043,Z 310.182,A -85,B 0,C 180,E1 15557.335,E2 15557.335} C_VEL
LIN {X 0,Y 450.641,Z 299.089,A -85,B 0,C 180,E1 15556.355,E2 15556.355} C_VEL
LIN {X 0,Y 443.632,Z 281.961,A -85,B 0,C 180,E1 15553.638,E2 15553.638} C_VEL
LIN {X 0,Y 436.782,Z 266.748,A -85,B 0,C 180,E1 15550.976,E2 15550.976} C_VEL
LIN {X 0,Y 434.457,Z 262.07,A -85,B 0,C 180,E1 15550.088,E2 15550.088} C_VEL
LIN {X 0,Y 433.262,Z 258.89,A -85,B 0,C 180,E1 15549.467,E2 15549.467} C_VEL
LIN {X 0,Y 433.248,Z 258.716,A -85,B 0,C 180,E1 15545.721,E2 15545.721} C_VEL
LIN {X 0,Y 433.259,Z 258.756,A -85,B 0,C 180,E1 15541.917,E2 15541.917} C_VEL
LIN {X 0,Y 433.257,Z 258.754,A -85,B 0,C 180,E1 15538.099,E2 15538.099} C_VEL
LIN {X 0,Y 433.253,Z 258.751,A -85,B 0,C 180,E1 15534.279,E2 15534.279} C_VEL
LIN {X 0,Y 433.253,Z 258.751,A -85,B 0,C 180,E1 15530.423,E2 15530.423} C_VEL
LIN {X 0,Y 433.242,Z 258.758,A -85,B 0,C 180,E1 15526.631,E2 15526.631} C_VEL
LIN {X 0,Y 433.238,Z 258.765,A -85,B 0,C 180,E1 15522.788,E2 15522.788} C_VEL
LIN {X 0,Y 433.241,Z 258.769,A -85,B 0,C 180,E1 15518.948,E2 15518.948} C_VEL
LIN {X 0,Y 433.248,Z 258.75,A -85,B 0,C 180,E1 15515.221,E2 15515.221} C_VEL
LIN {X 0,Y 433.259,Z 258.748,A -85,B 0,C 180,E1 15511.368,E2 15511.368} C_VEL
LIN {X 0,Y 433.26,Z 258.768,A -85,B 0,C 180,E1 15507.486,E2 15507.486} C_VEL
LIN {X 0,Y 433.259,Z 258.757,A -85,B 0,C 180,E1 15503.631,E2 15503.631} C_VEL
LIN {X 0,Y 433.253,Z 258.745,A -85,B 0,C 180,E1 15499.829,E2 15499.829} C_VEL
LIN {X 0,Y 433.241,Z 258.764,A -85,B 0,C 180,E1 15496.076,E2 15496.076} C_VEL
LIN {X 0,Y 433.234,Z 258.765,A -85,B 0,C 180,E1 15492.257,E2 15492.257} C_VEL
LIN {X 0,Y 433.234,Z 258.747,A -85,B 0,C 180,E1 15488.493,E2 15488.493} C_VEL
LIN {X 0,Y 433.249,Z 258.764,A -85,B 0,C 180,E1 15484.765,E2 15484.765} C_VEL
LIN {X 0,Y 433.26,Z 258.761,A -85,B 0,C 180,E1 15480.925,E2 15480.925} C_VEL
LIN {X 0,Y 433.256,Z 258.745,A -85,B 0,C 180,E1 15477.089,E2 15477.089} C_VEL
LIN {X 0,Y 433.261,Z 258.752,A -85,B 0,C 180,E1 15473.24,E2 15473.24} C_VEL
LIN {X 0,Y 433.252,Z 258.765,A -85,B 0,C 180,E1 15469.36,E2 15469.36} C_VEL
LIN {X 0,Y 433.24,Z 258.767,A -85,B 0,C 180,E1 15465.566,E2 15465.566} C_VEL
LIN {X 0,Y 433.232,Z 258.765,A -85,B 0,C 180,E1 15461.845,E2 15461.845} C_VEL
LIN {X 0,Y 433.232,Z 258.759,A -85,B 0,C 180,E1 15458.044,E2 15458.044} C_VEL
LIN {X 0,Y 433.246,Z 258.756,A -85,B 0,C 180,E1 15454.286,E2 15454.286} C_VEL
LIN {X 0,Y 433.261,Z 258.757,A -85,B 0,C 180,E1 15450.457,E2 15450.457} C_VEL
LIN {X 0,Y 433.261,Z 258.766,A -85,B 0,C 180,E1 15446.655,E2 15446.655} C_VEL
LIN {X 0,Y 433.259,Z 258.76,A -85,B 0,C 180,E1 15442.763,E2 15442.763} C_VEL
LIN {X 0,Y 433.278,Z 259.063,A -85,B 0,C 180,E1 15441.895,E2 15441.895} C_VEL
LIN {X 0,Y 434.733,Z 262.523,A -85,B 0,C 180,E1 15441.274,E2 15441.274} C_VEL
LIN {X 0,Y 435.882,Z 264.613,A -85,B 0,C 180,E1 15440.889,E2 15440.889} C_VEL
LIN {X 0,Y 442.336,Z 277.456,A -85,B 0,C 180,E1 15438.697,E2 15438.697} C_VEL
LIN {X 0,Y 449.868,Z 293.187,A -85,B 0,C 180,E1 15436.245,E2 15436.245} C_VEL
LIN {X 0,Y 454.174,Z 302.513,A -85,B 0,C 180,E1 15434.945,E2 15434.945} C_VEL
LIN {X 0,Y 462.77,Z 317.225,A -85,B 0,C 180,E1 15433.686,E2 15433.686} C_VEL
LIN {X 0,Y 465.024,Z 334.598,A -85,B 0,C 180,E1 15433.1,E2 15433.1} C_VEL
LIN {X 0,Y 459.759,Z 550.456,A -85,B 0,C 180,E1 15429.41,E2 15429.41} C_VEL
LIN {X 0,Y 458.314,Z 606.762,A -85,B 0,C 180,E1 15428.427,E2 15428.427} C_VEL
LIN {X 0,Y 456.946,Z 628.667,A -85,B 0,C 180,E1 15427.836,E2 15427.836} C_VEL
LIN {X 0,Y 455.216,Z 649.947,A -85,B 0,C 180,E1 15427.038,E2 15427.038} C_VEL
LIN {X 0,Y 453.267,Z 669.915,A -85,B 0,C 180,E1 15426.082,E2 15426.082} C_VEL
LIN {X 0,Y 450.981,Z 689.815,A -85,B 0,C 180,E1 15424.883,E2 15424.883} C_VEL
LIN {X 0,Y 448.437,Z 709.908,A -85,B 0,C 180,E1 15423.415,E2 15423.415} C_VEL
LIN {X 0,Y 445.928,Z 728.533,A -85,B 0,C 180,E1 15421.795,E2 15421.795} C_VEL
LIN {X 0,Y 443.428,Z 746.313,A -85,B 0,C 180,E1 15419.961,E2 15419.961} C_VEL
LIN {X 0,Y 440.984,Z 763.239,A -85,B 0,C 180,E1 15417.916,E2 15417.916} C_VEL
LIN {X 0,Y 438.749,Z 779.27,A -85,B 0,C 180,E1 15415.656,E2 15415.656} C_VEL
LIN {X 0,Y 436.87,Z 793.458,A -85,B 0,C 180,E1 15413.323,E2 15413.323} C_VEL
LIN {X 0,Y 435.241,Z 806.609,A -85,B 0,C 180,E1 15410.774,E2 15410.774} C_VEL
LIN {X 0,Y 433.925,Z 818.788,A -85,B 0,C 180,E1 15407.983,E2 15407.983} C_VEL
LIN {X 0,Y 433.038,Z 828.71,A -85,B 0,C 180,E1 15405.26,E2 15405.26} C_VEL
LIN {X 0,Y 432.457,Z 836.721,A -85,B 0,C 180,E1 15402.551,E2 15402.551} C_VEL
LIN {X 0,Y 432.13,Z 842.894,A -85,B 0,C 180,E1 15399.857,E2 15399.857} C_VEL
LIN {X 0,Y 431.98,Z 847.64,A -85,B 0,C 180,E1 15397.045,E2 15397.045} C_VEL
LIN {X 0,Y 431.917,Z 850.672,A -85,B 0,C 180,E1 15394.247,E2 15394.247} C_VEL
LIN {X 0,Y 431.901,Z 852.257,A -85,B 0,C 180,E1 15391.458,E2 15391.458} C_VEL
LIN {X 0,Y 431.909,Z 852.324,A -85,B 0,C 180,E1 15388.937,E2 15388.937} C_VEL
LIN {X 0,Y 431.912,Z 850.894,A -85,B 0,C 180,E1 15386.016,E2 15386.016} C_VEL
LIN {X 0,Y 431.957,Z 848.134,A -85,B 0,C 180,E1 15383.353,E2 15383.353} C_VEL
LIN {X 0,Y 432.106,Z 843.65,A -85,B 0,C 180,E1 15380.543,E2 15380.543} C_VEL
LIN {X 0,Y 432.381,Z 838.155,A -85,B 0,C 180,E1 15377.987,E2 15377.987} C_VEL
LIN {X 0,Y 432.889,Z 830.372,A -85,B 0,C 180,E1 15375.28,E2 15375.28} C_VEL
LIN {X 0,Y 433.711,Z 820.852,A -85,B 0,C 180,E1 15372.559,E2 15372.559} C_VEL
LIN {X 0,Y 434.847,Z 809.958,A -85,B 0,C 180,E1 15369.963,E2 15369.963} C_VEL
LIN {X 0,Y 436.305,Z 797.419,A -85,B 0,C 180,E1 15367.449,E2 15367.449} C_VEL
LIN {X 0,Y 438.236,Z 782.434,A -85,B 0,C 180,E1 15364.888,E2 15364.888} C_VEL
LIN {X 0,Y 440.305,Z 767.482,A -85,B 0,C 180,E1 15362.695,E2 15362.695} C_VEL
LIN {X 0,Y 442.66,Z 750.466,A -85,B 0,C 180,E1 15360.574,E2 15360.574} C_VEL
LIN {X 0,Y 445.157,Z 732.554,A -85,B 0,C 180,E1 15358.669,E2 15358.669} C_VEL
LIN {X 0,Y 447.677,Z 713.903,A -85,B 0,C 180,E1 15356.977,E2 15356.977} C_VEL
LIN {X 0,Y 450.039,Z 695.396,A -85,B 0,C 180,E1 15355.567,E2 15355.567} C_VEL
LIN {X 0,Y 452.332,Z 675.367,A -85,B 0,C 180,E1 15354.298,E2 15354.298} C_VEL
LIN {X 0,Y 454.45,Z 654.866,A -85,B 0,C 180,E1 15353.241,E2 15353.241} C_VEL
LIN {X 0,Y 456.222,Z 634.077,A -85,B 0,C 180,E1 15352.408,E2 15352.408} C_VEL
LIN {X 0,Y 457.675,Z 612.191,A -85,B 0,C 180,E1 15351.765,E2 15351.765} C_VEL
LIN {X 0,Y 458.6,Z 587.766,A -85,B 0,C 180,E1 15351.278,E2 15351.278} C_VEL
LIN {X 0,Y 463.838,Z 364.67,A -85,B 0,C 180,E1 15347.485,E2 15347.485} C_VEL
LIN {X 0,Y 464.468,Z 332.2,A -85,B 0,C 180,E1 15346.901,E2 15346.901} C_VEL
LIN {X 0,Y 462.13,Z 316.174,A -85,B 0,C 180,E1 15346.323,E2 15346.323} C_VEL
LIN {X 0,Y 453.617,Z 301.555,A -85,B 0,C 180,E1 15345.036,E2 15345.036} C_VEL
LIN {X 0,Y 445.909,Z 284.343,A -85,B 0,C 180,E1 15342.449,E2 15342.449} C_VEL
LIN {X 0,Y 439.546,Z 271.583,A -85,B 0,C 180,E1 15340.244,E2 15340.244} C_VEL
LIN {X 0,Y 436.996,Z 266.759,A -85,B 0,C 180,E1 15339.33,E2 15339.33} C_VEL
LIN {X 0,Y 435.178,Z 263.07,A -85,B 0,C 180,E1 15338.63,E2 15338.63} C_VEL
LIN {X 0,Y 433.441,Z 259.742,A -85,B 0,C 180,E1 15337.958,E2 15337.958} C_VEL
LIN {X 0,Y 433.263,Z 258.812,A -85,B 0,C 180,E1 15337.668,E2 15337.668} C_VEL
LIN {X 0,Y 433.256,Z 258.762,A -85,B 0,C 180,E1 15333.792,E2 15333.792} C_VEL
LIN {X 0,Y 433.261,Z 258.764,A -85,B 0,C 180,E1 15329.9,E2 15329.9} C_VEL
LIN {X 0,Y 433.253,Z 258.76,A -85,B 0,C 180,E1 15326.137,E2 15326.137} C_VEL
LIN {X 0,Y 433.254,Z 258.767,A -85,B 0,C 180,E1 15322.266,E2 15322.266} C_VEL
LIN {X 0,Y 433.256,Z 258.766,A -85,B 0,C 180,E1 15318.432,E2 15318.432} C_VEL
LIN {X 0,Y 433.261,Z 258.758,A -85,B 0,C 180,E1 15314.57,E2 15314.57} C_VEL
LIN {X 0,Y 433.249,Z 258.756,A -85,B 0,C 180,E1 15310.775,E2 15310.775} C_VEL
LIN {X 0,Y 433.237,Z 258.764,A -85,B 0,C 180,E1 15307.027,E2 15307.027} C_VEL
LIN {X 0,Y 433.229,Z 258.771,A -85,B 0,C 180,E1 15303.176,E2 15303.176} C_VEL
LIN {X 0,Y 433.224,Z 258.768,A -85,B 0,C 180,E1 15299.34,E2 15299.34} C_VEL
LIN {X 0,Y 433.231,Z 258.762,A -85,B 0,C 180,E1 15295.584,E2 15295.584} C_VEL
LIN {X 0,Y 433.252,Z 258.766,A -85,B 0,C 180,E1 15291.908,E2 15291.908} C_VEL
LIN {X 0,Y 433.257,Z 258.762,A -85,B 0,C 180,E1 15288.1,E2 15288.1} C_VEL
LIN {X 0,Y 433.244,Z 258.77,A -85,B 0,C 180,E1 15284.336,E2 15284.336} C_VEL
LIN {X 0,Y 433.256,Z 259.033,A -85,B 0,C 180,E1 15283.476,E2 15283.476} C_VEL
LIN {X 0,Y 434.62,Z 262.402,A -85,B 0,C 180,E1 15282.738,E2 15282.738} C_VEL
LIN {X 0,Y 435.613,Z 264.003,A -85,B 0,C 180,E1 15282.365,E2 15282.365} C_VEL
LIN {X 0,Y 441.555,Z 276.573,A -85,B 0,C 180,E1 15279.869,E2 15279.869} C_VEL
LIN {X 0,Y 447.92,Z 291.024,A -85,B 0,C 180,E1 15277.285,E2 15277.285} C_VEL
LIN {X 0,Y 451.85,Z 300.468,A -85,B 0,C 180,E1 15275.784,E2 15275.784} C_VEL
LIN {X 0,Y 458.891,Z 312.554,A -85,B 0,C 180,E1 15274.686,E2 15274.686} C_VEL
LIN {X 0,Y 461.965,Z 331.69,A -85,B 0,C 180,E1 15273.925,E2 15273.925} C_VEL
LIN {X 0,Y 454.966,Z 566.964,A -85,B 0,C 180,E1 15269.727,E2 15269.727} C_VEL
LIN {X 0,Y 453.772,Z 587.889,A -85,B 0,C 180,E1 15269.122,E2 15269.122} C_VEL
LIN {X 0,Y 452.28,Z 607.277,A -85,B 0,C 180,E1 15268.335,E2 15268.335} C_VEL
LIN {X 0,Y 450.379,Z 627.144,A -85,B 0,C 180,E1 15267.289,E2 15267.289} C_VEL
LIN {X 0,Y 448.219,Z 646.292,A -85,B 0,C 180,E1 15266.02,E2 15266.02} C_VEL
LIN {X 0,Y 445.987,Z 664.014,A -85,B 0,C 180,E1 15264.582,E2 15264.582} C_VEL
LIN {X 0,Y 443.651,Z 680.98,A -85,B 0,C 180,E1 15262.923,E2 15262.923} C_VEL
LIN {X 0,Y 441.365,Z 696.576,A -85,B 0,C 180,E1 15261.094,E2 15261.094} C_VEL
LIN {X 0,Y 439.237,Z 710.969,A -85,B 0,C 180,E1 15259.092,E2 15259.092} C_VEL
LIN {X 0,Y 437.834,Z 720.618,A -85,B 0,C 180,E1 15257.55,E2 15257.55} C_VEL
LIN {X 0,Y 436.233,Z 725.431,A -85,B 0,C 180,E1 15256.779,E2 15256.779} C_VEL
LIN {X 0,Y 428.934,Z 737.055,A -85,B 0,C 180,E1 15254.827,E2 15254.827} C_VEL
LIN {X 0,Y 427.439,Z 741.15,A -85,B 0,C 180,E1 15253.967,E2 15253.967} C_VEL
LIN {X 0,Y 426.117,Z 751.217,A -85,B 0,C 180,E1 15251.338,E2 15251.338} C_VEL
LIN {X 0,Y 425.197,Z 759.434,A -85,B 0,C 180,E1 15248.678,E2 15248.678} C_VEL
LIN {X 0,Y 424.602,Z 766.15,A -85,B 0,C 180,E1 15245.9,E2 15245.9} C_VEL
LIN {X 0,Y 424.282,Z 771.075,A -85,B 0,C 180,E1 15243.144,E2 15243.144} C_VEL
LIN {X 0,Y 424.136,Z 774.398,A -85,B 0,C 180,E1 15240.37,E2 15240.37} C_VEL
LIN {X 0,Y 424.087,Z 776.123,A -85,B 0,C 180,E1 15237.569,E2 15237.569} C_VEL
LIN {X 0,Y 424.078,Z 776.18,A -85,B 0,C 180,E1 15234.812,E2 15234.812} C_VEL
LIN {X 0,Y 424.116,Z 774.67,A -85,B 0,C 180,E1 15232.016,E2 15232.016} C_VEL
LIN {X 0,Y 424.225,Z 771.622,A -85,B 0,C 180,E1 15229.268,E2 15229.268} C_VEL
LIN {X 0,Y 424.499,Z 767.014,A -85,B 0,C 180,E1 15226.543,E2 15226.543} C_VEL
LIN {X 0,Y 425.024,Z 760.509,A -85,B 0,C 180,E1 15223.746,E2 15223.746} C_VEL
LIN {X 0,Y 425.846,Z 752.423,A -85,B 0,C 180,E1 15221.068,E2 15221.068} C_VEL
LIN {X 0,Y 427.026,Z 742.763,A -85,B 0,C 180,E1 15218.484,E2 15218.484} C_VEL
LIN {X 0,Y 428.554,Z 731.631,A -85,B 0,C 180,E1 15216.028,E2 15216.028} C_VEL
LIN {X 0,Y 430.399,Z 719.176,A -85,B 0,C 180,E1 15213.731,E2 15213.731} C_VEL
LIN {X 0,Y 432.508,Z 705.402,A -85,B 0,C 180,E1 15211.591,E2 15211.591} C_VEL
LIN {X 0,Y 434.819,Z 690.203,A -85,B 0,C 180,E1 15209.606,E2 15209.606} C_VEL
LIN {X 0,Y 437.243,Z 673.692,A -85,B 0,C 180,E1 15207.806,E2 15207.806} C_VEL
LIN {X 0,Y 439.617,Z 656.269,A -85,B 0,C 180,E1 15206.22,E2 15206.22} C_VEL
LIN {X 0,Y 441.978,Z 637.436,A -85,B 0,C 180,E1 15204.81,E2 15204.81} C_VEL
LIN {X 0,Y 444.019,Z 618.587,A -85,B 0,C 180,E1 15203.667,E2 15203.667} C_VEL
LIN {X 0,Y 445.835,Z 598.575,A -85,B 0,C 180,E1 15202.714,E2 15202.714} C_VEL
LIN {X 0,Y 447.275,Z 577.888,A -85,B 0,C 180,E1 15201.983,E2 15201.983} C_VEL
LIN {X 0,Y 448.235,Z 556.547,A -85,B 0,C 180,E1 15201.479,E2 15201.479} C_VEL
LIN {X 0,Y 454.562,Z 331.689,A -85,B 0,C 180,E1 15197.517,E2 15197.517} C_VEL
LIN {X 0,Y 451.389,Z 314.275,A -85,B 0,C 180,E1 15196.805,E2 15196.805} C_VEL
LIN {X 0,Y 442.696,Z 299.535,A -85,B 0,C 180,E1 15195.483,E2 15195.483} C_VEL
LIN {X 0,Y 435.901,Z 283.166,A -85,B 0,C 180,E1 15192.79,E2 15192.79} C_VEL
LIN {X 0,Y 428.852,Z 267.72,A -85,B 0,C 180,E1 15189.976,E2 15189.976} C_VEL
LIN {X 0,Y 426.511,Z 263.09,A -85,B 0,C 180,E1 15189.055,E2 15189.055} C_VEL
LIN {X 0,Y 425.338,Z 259.886,A -85,B 0,C 180,E1 15188.416,E2 15188.416} C_VEL
LIN {X 0,Y 425.309,Z 259.722,A -85,B 0,C 180,E1 15184.67,E2 15184.67} C_VEL
LIN {X 0,Y 425.306,Z 259.749,A -85,B 0,C 180,E1 15180.882,E2 15180.882} C_VEL
